C07314=1196.979,384.407,-79.887,-175.944,8.413,148.484
C07315=1196.984,384.160,-79.852,-175.945,8.410,148.484
C07316=1196.988,383.912,-79.818,-175.946,8.406,148.483
C07317=1196.992,383.664,-79.783,-175.947,8.404,148.483
C07318=1196.995,383.417,-79.748,-175.948,8.401,148.482
C07319=1197.000,383.170,-79.714,-175.948,8.397,148.481
C07320=1197.004,382.921,-79.679,-175.949,8.394,148.481
C07321=1197.007,382.674,-79.645,-175.950,8.392,148.480
C07322=1197.011,382.426,-79.610,-175.951,8.388,148.480
C07323=1197.016,382.179,-79.576,-175.952,8.385,148.479
C07324=1197.019,381.931,-79.541,-175.953,8.383,148.479
C07325=1197.024,381.684,-79.507,-175.954,8.379,148.478
C07326=1197.027,381.436,-79.471,-175.955,8.377,148.478
C07327=1197.031,381.189,-79.438,-175.956,8.374,148.477
C07328=1197.036,380.942,-79.403,-175.957,8.370,148.477
C07329=1197.040,380.693,-79.368,-175.958,8.368,148.476
C07330=1197.044,380.446,-79.334,-175.959,8.365,148.476
C07331=1197.048,380.198,-79.300,-175.960,8.362,148.475
C07332=1197.052,379.951,-79.265,-175.961,8.359,148.475
C07333=1197.055,379.703,-79.231,-175.962,8.356,148.474
C07334=1197.060,379.456,-79.196,-175.963,8.353,148.474
C07335=1197.065,379.208,-79.162,-175.965,8.349,148.473
C07336=1197.068,378.960,-79.128,-175.965,8.346,148.473
C07337=1197.072,378.713,-79.093,-175.967,8.343,148.472
C07338=1197.076,378.465,-79.058,-175.967,8.340,148.472
C07339=1197.080,378.218,-79.025,-175.969,8.337,148.471
C07340=1197.084,377.970,-78.990,-175.969,8.334,148.471
C07341=1197.088,377.722,-78.956,-175.971,8.331,148.470
C07342=1197.092,377.475,-78.921,-175.972,8.327,148.470
C07343=1197.096,377.227,-78.887,-175.973,8.325,148.469
C07344=1197.100,376.980,-78.853,-175.974,8.322,148.469
C07345=1197.104,376.732,-78.818,-175.975,8.319,148.468
C07346=1197.108,376.485,-78.784,-175.976,8.316,148.468
C07347=1197.113,376.237,-78.749,-175.978,8.312,148.467
C07348=1197.116,375.989,-78.716,-175.979,8.309,148.467
C07349=1197.121,375.741,-78.681,-175.980,8.306,148.467
C07350=1197.125,375.494,-78.648,-175.981,8.303,148.466
C07351=1197.129,375.246,-78.613,-175.983,8.300,148.466
C07352=1197.132,374.999,-78.579,-175.984,8.297,148.465
C07353=1197.136,374.751,-78.544,-175.985,8.294,148.465
C07354=1197.140,374.504,-78.510,-175.986,8.291,148.464
C07355=1197.145,374.256,-78.476,-175.988,8.287,148.464
C07356=1197.149,374.008,-78.442,-175.989,8.285,148.463
C07357=1197.153,373.760,-78.408,-175.990,8.281,148.463
C07358=1197.157,373.513,-78.374,-175.992,8.278,148.462
C07359=1197.161,373.265,-78.339,-175.993,8.275,148.462
C07360=1197.165,373.018,-78.306,-175.994,8.272,148.462
C07361=1197.169,372.770,-78.271,-175.995,8.268,148.461
C07362=1197.173,372.522,-78.237,-175.997,8.265,148.461
C07363=1197.177,372.275,-78.203,-175.998,8.263,148.460
C07364=1197.181,372.027,-78.170,-176.000,8.259,148.460
C07365=1197.185,371.779,-78.135,-176.001,8.256,148.459
C07366=1197.189,371.532,-78.101,-176.003,8.253,148.459
C07367=1197.194,371.285,-78.066,-176.003,8.249,148.458
C07368=1197.197,371.036,-78.033,-176.005,8.247,148.458
C07369=1197.201,370.789,-77.999,-176.006,8.243,148.457
C07370=1197.206,370.542,-77.965,-176.008,8.240,148.457
C07371=1197.210,370.294,-77.931,-176.009,8.237,148.457
C07372=1197.214,370.046,-77.897,-176.011,8.234,148.456
C07373=1197.218,369.799,-77.863,-176.012,8.231,148.456
C07374=1197.222,369.551,-77.829,-176.014,8.227,148.455
C07375=1197.226,369.303,-77.795,-176.015,8.225,148.455
C07376=1197.230,369.056,-77.761,-176.017,8.221,148.455
C07377=1197.234,368.808,-77.727,-176.018,8.218,148.454
C07378=1197.238,368.560,-77.693,-176.020,8.214,148.454
C07379=1197.242,368.312,-77.660,-176.021,8.212,148.453
C07380=1197.246,368.065,-77.625,-176.023,8.208,148.453
C07381=1197.250,367.818,-77.591,-176.024,8.205,148.453
C07382=1197.254,367.570,-77.558,-176.026,8.202,148.452
C07383=1197.258,367.322,-77.523,-176.027,8.199,148.452
C07384=1197.262,367.074,-77.490,-176.029,8.195,148.451
C07385=1197.267,366.793,-77.452,-176.030,8.192,148.451
C07386=1197.272,366.513,-77.413,-176.032,8.188,148.450
C07387=1197.277,366.232,-77.375,-176.034,8.184,148.450
C07388=1197.280,365.950,-77.337,-176.036,8.181,148.450
C07389=1197.285,365.703,-77.303,-176.037,8.178,148.449
C07390=1197.289,365.455,-77.270,-176.039,8.174,148.449
C07391=1197.293,365.208,-77.236,-176.040,8.172,148.449
C07392=1197.297,364.959,-77.202,-176.042,8.168,148.448
C07393=1197.301,364.712,-77.168,-176.044,8.164,148.448
C07394=1197.305,364.465,-77.135,-176.046,8.162,148.447
C07395=1197.309,364.217,-77.101,-176.048,8.158,148.447
C07396=1197.314,363.969,-77.067,-176.049,8.155,148.447
C07397=1197.317,363.721,-77.033,-176.051,8.152,148.446
C07398=1197.321,363.474,-77.000,-176.053,8.148,148.446
C07399=1197.325,363.226,-76.966,-176.054,8.146,148.446
C07400=1197.329,362.978,-76.933,-176.056,8.142,148.445
C07401=1197.334,362.731,-76.899,-176.057,8.140,148.445
C07402=1197.338,362.483,-76.866,-176.059,8.136,148.445
C07403=1197.342,362.235,-76.832,-176.061,8.132,148.444
C07404=1197.346,361.988,-76.798,-176.063,8.130,148.444
C07405=1197.350,361.740,-76.765,-176.064,8.126,148.443
C07406=1197.354,361.492,-76.732,-176.066,8.122,148.443
C07407=1197.358,361.245,-76.697,-176.068,8.120,148.443
C07408=1197.363,360.997,-76.664,-176.070,8.116,148.442
C07409=1197.366,360.749,-76.631,-176.071,8.113,148.442
C07410=1197.370,360.501,-76.598,-176.073,8.110,148.442
C07411=1197.374,360.254,-76.564,-176.075,8.107,148.441
C07412=1197.378,360.006,-76.531,-176.077,8.103,148.441
C07413=1197.382,359.758,-76.497,-176.078,8.100,148.441
C07414=1197.387,359.510,-76.464,-176.081,8.097,148.441
C07415=1197.391,359.263,-76.430,-176.082,8.093,148.440
C07416=1197.395,359.015,-76.396,-176.084,8.091,148.440
C07417=1197.399,358.767,-76.363,-176.086,8.087,148.439
C07418=1197.403,358.519,-76.330,-176.088,8.084,148.439
C07419=1197.407,358.272,-76.297,-176.089,8.081,148.439
C07420=1197.411,358.024,-76.264,-176.091,8.078,148.439
C07421=1197.415,357.776,-76.230,-176.093,8.074,148.438
C07422=1197.419,357.529,-76.197,-176.096,8.071,148.438
C07423=1197.424,357.281,-76.164,-176.097,8.068,148.438
C07424=1197.427,357.034,-76.130,-176.099,8.065,148.437
C07425=1197.431,356.786,-76.097,-176.101,8.061,148.437
C07426=1197.436,356.538,-76.064,-176.102,8.059,148.437
C07427=1197.440,356.291,-76.031,-176.105,8.055,148.437
C07428=1197.443,356.042,-75.997,-176.107,8.052,148.436
C07429=1197.447,355.794,-75.964,-176.109,8.048,148.436
C07430=1197.452,355.547,-75.931,-176.110,8.046,148.436
C07431=1197.456,355.299,-75.898,-176.113,8.042,148.435
C07432=1197.460,355.051,-75.865,-176.114,8.039,148.435
C07433=1197.464,354.803,-75.832,-176.116,8.036,148.435
C07434=1197.468,354.556,-75.798,-176.118,8.033,148.435
C07435=1197.472,354.308,-75.765,-176.120,8.029,148.434
C07436=1197.476,354.060,-75.732,-176.122,8.026,148.434
C07437=1197.481,353.813,-75.699,-176.124,8.024,148.434
C07438=1197.485,353.564,-75.666,-176.126,8.020,148.433
C07439=1197.489,353.316,-75.633,-176.128,8.017,148.433
C07440=1197.493,353.069,-75.600,-176.130,8.013,148.433
C07441=1197.497,352.821,-75.567,-176.132,8.011,148.433
C07442=1197.502,352.573,-75.534,-176.134,8.007,148.432
C07443=1197.506,352.326,-75.501,-176.136,8.004,148.432
C07444=1197.509,352.078,-75.468,-176.138,8.001,148.432
C07445=1197.513,351.830,-75.435,-176.140,7.998,148.432
C07446=1197.518,351.582,-75.403,-176.142,7.995,148.431
C07447=1197.522,351.334,-75.369,-176.144,7.991,148.431
C07448=1197.526,351.087,-75.336,-176.145,7.988,148.431
C07449=1197.530,350.839,-75.303,-176.148,7.985,148.431
C07450=1197.534,350.591,-75.270,-176.150,7.982,148.430
C07451=1197.539,350.343,-75.237,-176.152,7.978,148.430
C07452=1197.542,350.095,-75.205,-176.154,7.976,148.430
C07453=1197.546,349.848,-75.172,-176.156,7.972,148.430
C07454=1197.550,349.600,-75.139,-176.158,7.969,148.429
C07455=1197.555,349.352,-75.107,-176.160,7.966,148.429
C07456=1197.560,349.104,-75.073,-176.162,7.963,148.429
C07457=1197.563,348.857,-75.041,-176.164,7.960,148.429
C07458=1197.567,348.609,-75.008,-176.166,7.956,148.428
C07459=1197.571,348.361,-74.975,-176.168,7.954,148.428
C07460=1197.576,348.113,-74.942,-176.170,7.951,148.428
C07461=1197.580,347.865,-74.910,-176.172,7.947,148.428
C07462=1197.583,347.617,-74.877,-176.175,7.944,148.428
C07463=1197.588,347.370,-74.844,-176.176,7.941,148.427
C07464=1197.592,347.121,-74.811,-176.178,7.938,148.427
C07465=1197.596,346.874,-74.778,-176.180,7.934,148.427
C07466=1197.601,346.626,-74.747,-176.182,7.931,148.427
C07467=1197.605,346.379,-74.714,-176.184,7.929,148.426
C07468=1197.609,346.130,-74.681,-176.186,7.925,148.426
C07469=1197.612,345.883,-74.649,-176.189,7.922,148.426
C07470=1197.617,345.635,-74.615,-176.191,7.919,148.426
C07471=1197.621,345.387,-74.583,-176.192,7.916,148.426
C07472=1197.625,345.139,-74.550,-176.195,7.913,148.425
C07473=1197.630,344.892,-74.518,-176.197,7.909,148.425
C07474=1197.634,344.644,-74.485,-176.199,7.906,148.425
C07475=1197.638,344.396,-74.453,-176.201,7.904,148.425
C07476=1197.642,344.148,-74.421,-176.203,7.900,148.424
C07477=1197.646,343.900,-74.388,-176.206,7.897,148.424
C07478=1197.650,343.651,-74.355,-176.208,7.894,148.424
C07479=1197.654,343.405,-74.323,-176.210,7.891,148.424
C07480=1197.659,343.156,-74.291,-176.212,7.888,148.424
C07481=1197.662,342.909,-74.258,-176.214,7.885,148.424
C07482=1197.667,342.661,-74.226,-176.216,7.881,148.423
C07483=1197.671,342.412,-74.193,-176.218,7.879,148.423
C07484=1197.675,342.165,-74.161,-176.220,7.876,148.423
C07485=1197.680,341.917,-74.129,-176.222,7.872,148.423
C07486=1197.683,341.669,-74.097,-176.225,7.869,148.423
C07487=1197.687,341.421,-74.064,-176.227,7.867,148.423
C07488=1197.692,341.173,-74.031,-176.229,7.863,148.422
C07489=1197.697,340.895,-73.995,-176.231,7.860,148.422
C07490=1197.701,340.617,-73.958,-176.234,7.857,148.422
C07491=1197.706,340.338,-73.923,-176.236,7.853,148.422
C07492=1197.710,340.060,-73.887,-176.239,7.849,148.421
C07493=1197.715,339.812,-73.855,-176.241,7.846,148.421
C07494=1197.718,339.564,-73.822,-176.243,7.844,148.421
C07495=1197.723,339.316,-73.790,-176.245,7.840,148.421
C07496=1197.726,339.068,-73.758,-176.247,7.837,148.421
C07497=1197.731,338.820,-73.726,-176.250,7.834,148.421
C07498=1197.735,338.572,-73.694,-176.252,7.832,148.421
C07499=1197.739,338.324,-73.661,-176.254,7.828,148.420
C07500=1197.744,338.077,-73.629,-176.256,7.825,148.420
C07501=1197.748,337.829,-73.597,-176.258,7.822,148.420
C07502=1197.752,337.581,-73.565,-176.260,7.819,148.420
C07503=1197.756,337.332,-73.532,-176.263,7.816,148.420
C07504=1197.761,337.085,-73.501,-176.265,7.813,148.420
C07505=1197.765,336.837,-73.469,-176.267,7.809,148.419
C07506=1197.768,336.589,-73.436,-176.269,7.807,148.419
C07507=1197.772,336.341,-73.404,-176.272,7.804,148.419
C07508=1197.777,336.094,-73.372,-176.274,7.800,148.419
C07509=1197.781,335.846,-73.340,-176.276,7.797,148.419
C07510=1197.785,335.597,-73.308,-176.278,7.795,148.419
C07511=1197.790,335.350,-73.276,-176.280,7.792,148.419
C07512=1197.793,335.102,-73.244,-176.283,7.788,148.418
C07513=1197.798,334.853,-73.212,-176.285,7.785,148.418
C07514=1197.802,334.606,-73.181,-176.287,7.783,148.418
C07515=1197.806,334.358,-73.149,-176.289,7.779,148.418
C07516=1197.810,334.110,-73.116,-176.291,7.776,148.418
C07517=1197.815,333.862,-73.085,-176.294,7.773,148.418
C07518=1197.818,333.614,-73.053,-176.296,7.771,148.418
C07519=1197.823,333.366,-73.020,-176.298,7.768,148.418
C07520=1197.827,333.119,-72.989,-176.301,7.764,148.417
C07521=1197.831,332.870,-72.958,-176.303,7.761,148.417
C07522=1197.836,332.622,-72.926,-176.305,7.759,148.417
C07523=1197.840,332.374,-72.894,-176.307,7.755,148.417
C07524=1197.843,332.126,-72.862,-176.310,7.752,148.417
C07525=1197.848,331.879,-72.831,-176.312,7.749,148.417
C07526=1197.852,331.631,-72.798,-176.314,7.746,148.417
C07527=1197.856,331.383,-72.766,-176.317,7.743,148.417
C07528=1197.861,331.135,-72.736,-176.319,7.740,148.416
C07529=1197.864,330.887,-72.704,-176.321,7.737,148.416
C07530=1197.869,330.639,-72.672,-176.323,7.735,148.416
C07531=1197.873,330.391,-72.640,-176.325,7.731,148.416
C07532=1197.877,330.144,-72.608,-176.328,7.728,148.416
C07533=1197.881,329.895,-72.577,-176.330,7.725,148.416
C07534=1197.885,329.647,-72.545,-176.332,7.722,148.416
C07535=1197.890,329.399,-72.513,-176.335,7.719,148.416
C07536=1197.894,329.151,-72.481,-176.337,7.716,148.415
C07537=1197.898,328.903,-72.451,-176.340,7.713,148.415
C07538=1197.902,328.655,-72.419,-176.341,7.711,148.415
C07539=1197.906,328.408,-72.387,-176.344,7.708,148.415
C07540=1197.910,328.159,-72.356,-176.346,7.704,148.415
C07541=1197.915,327.912,-72.324,-176.349,7.701,148.415
C07542=1197.919,327.663,-72.292,-176.351,7.699,148.415
C07543=1197.923,327.415,-72.261,-176.353,7.696,148.415
C07544=1197.927,327.167,-72.230,-176.355,7.692,148.415
C07545=1197.931,326.919,-72.199,-176.358,7.690,148.415
C07546=1197.936,326.671,-72.167,-176.360,7.687,148.414
C07547=1197.939,326.423,-72.135,-176.363,7.684,148.414
C07548=1197.944,326.175,-72.104,-176.365,7.680,148.414
C07549=1197.948,325.927,-72.073,-176.367,7.678,148.414
C07550=1197.952,325.679,-72.042,-176.369,7.675,148.414
C07551=1197.957,325.431,-72.009,-176.372,7.672,148.414
C07552=1197.961,325.183,-71.979,-176.374,7.669,148.414
C07553=1197.965,324.935,-71.947,-176.376,7.666,148.414
C07554=1197.970,324.687,-71.916,-176.378,7.663,148.414
C07555=1197.974,324.439,-71.884,-176.381,7.660,148.414
C07556=1197.978,324.191,-71.853,-176.384,7.657,148.414
C07557=1197.982,323.943,-71.822,-176.385,7.654,148.414
C07558=1197.986,323.695,-71.791,-176.388,7.651,148.414
C07559=1197.991,323.448,-71.759,-176.390,7.648,148.413
C07560=1197.995,323.199,-71.728,-176.393,7.645,148.413
C07561=1197.999,322.952,-71.697,-176.395,7.643,148.413
C07562=1198.003,322.703,-71.666,-176.397,7.640,148.413
C07563=1198.008,322.455,-71.635,-176.400,7.637,148.413
C07564=1198.011,322.208,-71.604,-176.402,7.633,148.413
C07565=1198.015,321.960,-71.573,-176.404,7.631,148.413
C07566=1198.019,321.711,-71.542,-176.407,7.628,148.413
C07567=1198.024,321.464,-71.510,-176.409,7.625,148.413
C07568=1198.028,321.216,-71.479,-176.412,7.622,148.413
C07569=1198.032,320.967,-71.448,-176.414,7.619,148.413
C07570=1198.037,320.720,-71.417,-176.416,7.616,148.413
C07571=1198.041,320.471,-71.386,-176.419,7.613,148.413
C07572=1198.045,320.223,-71.355,-176.421,7.611,148.413
C07573=1198.050,319.975,-71.324,-176.424,7.608,148.413
C07574=1198.053,319.727,-71.292,-176.426,7.604,148.412
C07575=1198.057,319.479,-71.262,-176.428,7.601,148.412
C07576=1198.061,319.231,-71.231,-176.431,7.599,148.412
C07577=1198.066,318.983,-71.200,-176.433,7.596,148.412
C07578=1198.070,318.735,-71.169,-176.436,7.593,148.412
C07579=1198.074,318.487,-71.138,-176.438,7.590,148.412
C07580=1198.079,318.239,-71.107,-176.440,7.587,148.412
C07581=1198.083,317.991,-71.077,-176.443,7.584,148.412
C07582=1198.087,317.742,-71.046,-176.445,7.581,148.412
C07583=1198.091,317.494,-71.015,-176.447,7.579,148.412
C07584=1198.096,317.247,-70.983,-176.450,7.576,148.412
C07585=1198.100,316.998,-70.952,-176.452,7.573,148.412
C07586=1198.104,316.751,-70.922,-176.455,7.570,148.412
C07587=1198.108,316.503,-70.891,-176.457,7.567,148.412
C07588=1198.112,316.254,-70.860,-176.459,7.564,148.412
C07589=1198.117,316.006,-70.829,-176.462,7.561,148.412
C07590=1198.121,315.759,-70.799,-176.464,7.558,148.412
C07591=1198.125,315.510,-70.768,-176.466,7.555,148.412
C07592=1198.129,315.262,-70.737,-176.469,7.552,148.412
C07593=1198.134,314.986,-70.703,-176.472,7.549,148.412
C07594=1198.139,314.709,-70.669,-176.475,7.546,148.412
C07595=1198.143,314.433,-70.635,-176.477,7.543,148.411
C07596=1198.148,314.158,-70.601,-176.479,7.540,148.411
C07597=1198.152,313.909,-70.569,-176.482,7.537,148.411
C07598=1198.157,313.660,-70.539,-176.485,7.534,148.411
C07599=1198.161,313.413,-70.509,-176.487,7.531,148.411
C07600=1198.166,313.165,-70.478,-176.489,7.528,148.411
C07601=1198.170,312.916,-70.447,-176.492,7.525,148.411
C07602=1198.173,312.668,-70.417,-176.495,7.522,148.411
C07603=1198.178,312.420,-70.386,-176.497,7.520,148.411
C07604=1198.182,312.173,-70.356,-176.499,7.517,148.411
C07605=1198.186,311.924,-70.325,-176.502,7.514,148.411
C07606=1198.191,311.676,-70.294,-176.504,7.512,148.411
C07607=1198.195,311.428,-70.265,-176.506,7.509,148.411
C07608=1198.199,311.180,-70.234,-176.509,7.506,148.411
C07609=1198.203,310.931,-70.203,-176.511,7.502,148.411
C07610=1198.207,310.684,-70.173,-176.514,7.500,148.411
C07611=1198.212,310.436,-70.142,-176.516,7.497,148.411
C07612=1198.216,310.187,-70.113,-176.519,7.494,148.411
C07613=1198.221,309.939,-70.082,-176.521,7.492,148.411
C07614=1198.225,309.692,-70.052,-176.523,7.489,148.411
C07615=1198.229,309.443,-70.021,-176.526,7.486,148.411
C07616=1198.233,309.195,-69.991,-176.528,7.483,148.411
C07617=1198.237,308.947,-69.960,-176.531,7.480,148.411
C07618=1198.242,308.699,-69.930,-176.533,7.477,148.411
C07619=1198.246,308.451,-69.900,-176.536,7.474,148.411
C07620=1198.251,308.203,-69.869,-176.538,7.472,148.411
C07621=1198.254,307.954,-69.839,-176.541,7.469,148.411
C07622=1198.259,307.706,-69.809,-176.543,7.466,148.411
C07623=1198.263,307.458,-69.779,-176.545,7.464,148.411
C07624=1198.267,307.210,-69.748,-176.548,7.461,148.411
C07625=1198.272,306.962,-69.718,-176.551,7.458,148.411
C07626=1198.276,306.714,-69.688,-176.553,7.455,148.411
C07627=1198.280,306.466,-69.658,-176.555,7.452,148.411
C07628=1198.284,306.217,-69.628,-176.558,7.449,148.411
C07629=1198.289,305.969,-69.598,-176.560,7.447,148.411
C07630=1198.292,305.721,-69.567,-176.563,7.444,148.411
C07631=1198.297,305.473,-69.537,-176.565,7.441,148.411
C07632=1198.301,305.225,-69.507,-176.568,7.439,148.411
C07633=1198.306,304.976,-69.477,-176.570,7.436,148.411
C07634=1198.310,304.729,-69.447,-176.573,7.433,148.411
C07635=1198.314,304.480,-69.418,-176.576,7.430,148.411
C07636=1198.319,304.232,-69.387,-176.577,7.427,148.411
C07637=1198.323,303.984,-69.357,-176.580,7.424,148.411
C07638=1198.327,303.737,-69.327,-176.583,7.421,148.411
C07639=1198.332,303.488,-69.297,-176.585,7.419,148.411
C07640=1198.335,303.240,-69.267,-176.587,7.416,148.411
C07641=1198.340,302.991,-69.236,-176.590,7.413,148.411
C07642=1198.344,302.743,-69.207,-176.592,7.411,148.411
C07643=1198.348,302.495,-69.177,-176.595,7.408,148.411
C07644=1198.353,302.247,-69.147,-176.598,7.405,148.411
C07645=1198.357,301.998,-69.117,-176.600,7.402,148.411
C07646=1198.361,301.751,-69.087,-176.603,7.399,148.411
C07647=1198.365,301.502,-69.058,-176.605,7.396,148.411
C07648=1198.370,301.254,-69.028,-176.607,7.394,148.411
C07649=1198.374,301.006,-68.998,-176.610,7.391,148.411
C07650=1198.378,300.758,-68.968,-176.612,7.388,148.411
C07651=1198.382,300.510,-68.939,-176.614,7.386,148.411
C07652=1198.387,300.262,-68.908,-176.617,7.383,148.411
C07653=1198.391,300.013,-68.878,-176.620,7.380,148.411
C07654=1198.395,299.765,-68.849,-176.622,7.377,148.411
C07655=1198.400,299.517,-68.819,-176.625,7.374,148.411
C07656=1198.404,299.269,-68.789,-176.627,7.372,148.411
C07657=1198.408,299.021,-68.759,-176.630,7.369,148.411
C07658=1198.413,298.772,-68.730,-176.632,7.366,148.411
C07659=1198.417,298.524,-68.700,-176.634,7.364,148.411
C07660=1198.421,298.276,-68.671,-176.637,7.361,148.411
C07661=1198.426,298.027,-68.641,-176.640,7.358,148.411
C07662=1198.430,297.780,-68.611,-176.642,7.356,148.412
C07663=1198.434,297.531,-68.581,-176.645,7.353,148.412
C07664=1198.438,297.283,-68.552,-176.647,7.350,148.412
C07665=1198.443,297.035,-68.523,-176.649,7.348,148.412
C07666=1198.447,296.787,-68.493,-176.652,7.345,148.412
C07667=1198.451,296.539,-68.464,-176.655,7.342,148.412
C07668=1198.456,296.290,-68.434,-176.657,7.339,148.412
C07669=1198.460,296.042,-68.404,-176.660,7.336,148.412
C07670=1198.465,295.794,-68.375,-176.662,7.334,148.412
C07671=1198.469,295.546,-68.345,-176.665,7.331,148.412
C07672=1198.473,295.297,-68.316,-176.667,7.328,148.412
C07673=1198.477,295.049,-68.286,-176.669,7.326,148.412
C07674=1198.481,294.801,-68.257,-176.672,7.323,148.412
C07675=1198.485,294.552,-68.228,-176.675,7.320,148.412
C07676=1198.490,294.304,-68.198,-176.677,7.318,148.412
C07677=1198.494,294.057,-68.169,-176.680,7.315,148.412
C07678=1198.499,293.808,-68.140,-176.683,7.312,148.412
C07679=1198.503,293.560,-68.110,-176.685,7.310,148.412
C07680=1198.507,293.312,-68.081,-176.688,7.307,148.412
C07681=1198.511,293.064,-68.051,-176.690,7.305,148.412
C07682=1198.515,292.815,-68.022,-176.692,7.302,148.413
C07683=1198.519,292.567,-67.992,-176.695,7.299,148.413
C07684=1198.524,292.319,-67.963,-176.697,7.296,148.413
C07685=1198.529,292.071,-67.934,-176.700,7.293,148.413
C07686=1198.533,291.822,-67.905,-176.702,7.291,148.413
C07687=1198.537,291.574,-67.876,-176.705,7.288,148.413
C07688=1198.541,291.326,-67.846,-176.708,7.285,148.413
C07689=1198.545,291.078,-67.817,-176.710,7.283,148.413
C07690=1198.550,290.829,-67.788,-176.712,7.280,148.413
C07691=1198.555,290.581,-67.759,-176.715,7.277,148.413
C07692=1198.559,290.333,-67.729,-176.717,7.275,148.413
C07693=1198.563,290.085,-67.700,-176.720,7.272,148.413
C07694=1198.567,289.836,-67.670,-176.723,7.270,148.413
C07695=1198.572,289.587,-67.642,-176.725,7.267,148.413
C07696=1198.577,289.340,-67.613,-176.728,7.264,148.413
C07697=1198.581,289.065,-67.581,-176.731,7.261,148.413
C07698=1198.585,288.791,-67.548,-176.733,7.258,148.413
C07699=1198.590,288.517,-67.517,-176.736,7.256,148.414
C07700=1198.596,288.242,-67.484,-176.739,7.253,148.414
C07701=1198.600,287.994,-67.455,-176.741,7.250,148.414
C07702=1198.603,287.746,-67.426,-176.744,7.247,148.414
C07703=1198.608,287.497,-67.397,-176.746,7.245,148.414
C07704=1198.612,287.249,-67.368,-176.749,7.242,148.414
C07705=1198.617,287.000,-67.340,-176.751,7.240,148.414
C07706=1198.621,286.752,-67.310,-176.754,7.237,148.414
C07707=1198.625,286.505,-67.282,-176.757,7.234,148.414
C07708=1198.630,286.256,-67.253,-176.759,7.232,148.414
C07709=1198.634,286.008,-67.223,-176.762,7.229,148.414
C07710=1198.638,285.759,-67.195,-176.764,7.227,148.414
C07711=1198.643,285.511,-67.166,-176.767,7.224,148.414
C07712=1198.647,285.263,-67.137,-176.769,7.221,148.414
C07713=1198.651,285.014,-67.108,-176.771,7.218,148.414
C07714=1198.656,284.766,-67.080,-176.775,7.216,148.415
C07715=1198.660,284.518,-67.050,-176.777,7.213,148.415
C07716=1198.664,284.269,-67.022,-176.779,7.210,148.415
C07717=1198.668,284.021,-66.993,-176.782,7.208,148.415
C07718=1198.673,283.773,-66.964,-176.784,7.205,148.415
C07719=1198.678,283.525,-66.935,-176.786,7.203,148.415
C07720=1198.681,283.276,-66.907,-176.790,7.200,148.415
C07721=1198.686,283.028,-66.878,-176.792,7.197,148.415
C07722=1198.691,282.780,-66.849,-176.794,7.195,148.415
C07723=1198.694,282.531,-66.821,-176.797,7.192,148.415
C07724=1198.699,282.283,-66.792,-176.799,7.190,148.415
C07725=1198.704,282.035,-66.763,-176.802,7.187,148.415
C07726=1198.708,281.787,-66.735,-176.805,7.185,148.416
C07727=1198.712,281.538,-66.706,-176.807,7.182,148.416
C07728=1198.717,281.290,-66.677,-176.810,7.179,148.416
C07729=1198.721,281.042,-66.649,-176.812,7.177,148.416
C07730=1198.725,280.793,-66.620,-176.815,7.174,148.416
C07731=1198.729,280.545,-66.591,-176.817,7.172,148.416
C07732=1198.734,280.297,-66.563,-176.820,7.169,148.416
C07733=1198.738,280.048,-66.534,-176.822,7.167,148.416
C07734=1198.743,279.800,-66.507,-176.825,7.164,148.416
C07735=1198.747,279.552,-66.477,-176.827,7.162,148.416
C07736=1198.751,279.303,-66.449,-176.830,7.159,148.417
C07737=1198.756,279.055,-66.421,-176.832,7.157,148.417
C07738=1198.760,278.806,-66.392,-176.835,7.154,148.417
C07739=1198.765,278.558,-66.364,-176.837,7.152,148.417
C07740=1198.769,278.310,-66.335,-176.840,7.149,148.417
C07741=1198.773,278.061,-66.307,-176.843,7.146,148.417
C07742=1198.778,277.813,-66.278,-176.845,7.144,148.417
C07743=1198.781,277.565,-66.250,-176.848,7.141,148.417
C07744=1198.787,277.316,-66.222,-176.850,7.139,148.417
C07745=1198.790,277.068,-66.193,-176.853,7.136,148.418
C07746=1198.795,276.820,-66.165,-176.856,7.134,148.418
C07747=1198.799,276.571,-66.137,-176.858,7.131,148.418
C07748=1198.804,276.323,-66.108,-176.860,7.128,148.418
C07749=1198.808,276.075,-66.080,-176.864,7.126,148.418
C07750=1198.811,275.826,-66.052,-176.866,7.124,148.418
C07751=1198.816,275.578,-66.023,-176.868,7.121,148.418
C07752=1198.820,275.330,-65.995,-176.871,7.118,148.418
C07753=1198.825,275.081,-65.967,-176.874,7.116,148.418
C07754=1198.829,274.833,-65.939,-176.876,7.114,148.419
C07755=1198.834,274.585,-65.910,-176.879,7.111,148.419
C07756=1198.838,274.336,-65.882,-176.881,7.108,148.419
C07757=1198.842,274.088,-65.854,-176.884,7.106,148.419
C07758=1198.847,273.839,-65.826,-176.886,7.104,148.419
C07759=1198.851,273.591,-65.798,-176.889,7.100,148.419
C07760=1198.856,273.342,-65.770,-176.891,7.098,148.419
C07761=1198.860,273.094,-65.742,-176.894,7.096,148.419
C07762=1198.864,272.845,-65.714,-176.896,7.093,148.419
C07763=1198.869,272.597,-65.685,-176.899,7.090,148.419
C07764=1198.873,272.349,-65.658,-176.901,7.088,148.420
C07765=1198.877,272.101,-65.630,-176.904,7.086,148.420
C07766=1198.882,271.853,-65.601,-176.906,7.083,148.420
C07767=1198.886,271.604,-65.573,-176.909,7.080,148.420
C07768=1198.891,271.355,-65.546,-176.912,7.079,148.420
C07769=1198.895,271.107,-65.517,-176.914,7.076,148.420
C07770=1198.900,270.859,-65.489,-176.917,7.073,148.420
C07771=1198.903,270.610,-65.461,-176.920,7.071,148.421
C07772=1198.908,270.362,-65.433,-176.922,7.068,148.421
C07773=1198.913,270.113,-65.406,-176.925,7.065,148.421
C07774=1198.917,269.865,-65.378,-176.927,7.063,148.421
C07775=1198.921,269.617,-65.350,-176.930,7.061,148.421
C07776=1198.926,269.368,-65.321,-176.932,7.058,148.421
C07777=1198.930,269.120,-65.294,-176.935,7.055,148.421
C07778=1198.935,268.872,-65.266,-176.937,7.054,148.421
C07779=1198.938,268.623,-65.238,-176.940,7.051,148.422
C07780=1198.944,268.374,-65.211,-176.942,7.048,148.422
C07781=1198.948,268.127,-65.183,-176.945,7.047,148.422
C07782=1198.952,267.878,-65.155,-176.948,7.044,148.422
C07783=1198.957,267.629,-65.128,-176.950,7.041,148.422
C07784=1198.960,267.381,-65.099,-176.953,7.039,148.422
C07785=1198.965,267.133,-65.071,-176.955,7.037,148.422
C07786=1198.970,266.884,-65.044,-176.958,7.034,148.422
C07787=1198.974,266.636,-65.016,-176.960,7.032,148.423
C07788=1198.978,266.387,-64.989,-176.963,7.029,148.423
C07789=1198.983,266.139,-64.961,-176.965,7.026,148.423
C07790=1198.987,265.891,-64.933,-176.968,7.024,148.423
C07791=1198.991,265.642,-64.906,-176.971,7.022,148.423
C07792=1198.996,265.394,-64.877,-176.973,7.019,148.423
C07793=1199.000,265.145,-64.850,-176.976,7.017,148.424
C07794=1199.005,264.897,-64.822,-176.978,7.015,148.424
C07795=1199.009,264.648,-64.795,-176.981,7.012,148.424
C07796=1199.014,264.401,-64.767,-176.983,7.010,148.424
C07797=1199.018,264.151,-64.740,-176.986,7.007,148.424
C07798=1199.022,263.903,-64.712,-176.988,7.005,148.424
C07799=1199.027,263.655,-64.685,-176.991,7.002,148.424
C07800=1199.031,263.406,-64.658,-176.994,7.000,148.424
C07801=1199.036,263.133,-64.627,-176.997,6.997,148.425
C07802=1199.041,262.861,-64.597,-176.999,6.995,148.425
C07803=1199.045,262.587,-64.567,-177.002,6.992,148.425
C07804=1199.051,262.315,-64.537,-177.005,6.989,148.425
C07805=1199.055,262.067,-64.509,-177.007,6.987,148.425
C07806=1199.059,261.818,-64.481,-177.010,6.984,148.425
C07807=1199.064,261.569,-64.454,-177.012,6.982,148.426
C07808=1199.068,261.321,-64.427,-177.015,6.979,148.426
C07809=1199.073,261.073,-64.400,-177.018,6.977,148.426
C07810=1199.077,260.824,-64.372,-177.020,6.974,148.426
C07811=1199.081,260.576,-64.344,-177.023,6.972,148.426
C07812=1199.086,260.327,-64.317,-177.025,6.970,148.426
C07813=1199.090,260.079,-64.290,-177.028,6.968,148.427
C07814=1199.095,259.830,-64.263,-177.030,6.965,148.427
C07815=1199.099,259.582,-64.235,-177.033,6.962,148.427
C07816=1199.103,259.333,-64.208,-177.036,6.961,148.427
C07817=1199.108,259.085,-64.181,-177.038,6.958,148.427
C07818=1199.113,258.836,-64.154,-177.041,6.956,148.427
C07819=1199.117,258.588,-64.127,-177.043,6.953,148.427
C07820=1199.120,258.340,-64.099,-177.046,6.951,148.428
C07821=1199.125,258.091,-64.072,-177.049,6.949,148.428
C07822=1199.130,257.843,-64.045,-177.051,6.946,148.428
C07823=1199.134,257.594,-64.018,-177.054,6.944,148.428
C07824=1199.139,257.346,-63.991,-177.056,6.942,148.428
C07825=1199.144,257.097,-63.964,-177.059,6.939,148.429
C07826=1199.147,256.848,-63.936,-177.061,6.937,148.429
C07827=1199.151,256.600,-63.909,-177.064,6.935,148.429
C07828=1199.156,256.352,-63.882,-177.067,6.932,148.429
C07829=1199.161,256.103,-63.855,-177.069,6.930,148.429
C07830=1199.165,255.855,-63.828,-177.072,6.928,148.429
C07831=1199.170,255.606,-63.801,-177.074,6.925,148.429
C07832=1199.175,255.358,-63.774,-177.077,6.923,148.430
C07833=1199.178,255.109,-63.747,-177.080,6.920,148.430
C07834=1199.183,254.860,-63.720,-177.082,6.918,148.430
C07835=1199.187,254.612,-63.693,-177.084,6.916,148.430
C07836=1199.192,254.363,-63.666,-177.087,6.913,148.430
C07837=1199.196,254.115,-63.640,-177.090,6.911,148.431
C07838=1199.200,253.867,-63.612,-177.092,6.909,148.431
C07839=1199.205,253.618,-63.585,-177.095,6.906,148.431
C07840=1199.210,253.370,-63.558,-177.097,6.904,148.431
C07841=1199.214,253.122,-63.532,-177.100,6.902,148.431
C07842=1199.218,252.872,-63.504,-177.103,6.899,148.431
C07843=1199.222,252.624,-63.477,-177.105,6.897,148.432
C07844=1199.227,252.375,-63.450,-177.108,6.894,148.432
C07845=1199.231,252.127,-63.424,-177.111,6.893,148.432
C07846=1199.236,251.879,-63.397,-177.113,6.890,148.432
C07847=1199.241,251.630,-63.370,-177.116,6.888,148.432
C07848=1199.245,251.381,-63.344,-177.118,6.886,148.432
C07849=1199.249,251.133,-63.317,-177.121,6.884,148.433
C07850=1199.254,250.884,-63.290,-177.123,6.881,148.433
C07851=1199.258,250.636,-63.263,-177.126,6.879,148.433
C07852=1199.262,250.388,-63.236,-177.128,6.877,148.433
C07853=1199.267,250.139,-63.210,-177.131,6.874,148.433
C07854=1199.271,249.890,-63.184,-177.133,6.872,148.434
C07855=1199.276,249.642,-63.156,-177.136,6.870,148.434
C07856=1199.281,249.393,-63.129,-177.139,6.867,148.434
C07857=1199.285,249.145,-63.103,-177.141,6.865,148.434
C07858=1199.289,248.896,-63.077,-177.144,6.863,148.434
C07859=1199.293,248.648,-63.050,-177.146,6.860,148.434
C07860=1199.298,248.399,-63.023,-177.149,6.858,148.435
C07861=1199.303,248.150,-62.997,-177.151,6.856,148.435
C07862=1199.307,247.902,-62.970,-177.154,6.853,148.435
C07863=1199.312,247.654,-62.943,-177.156,6.851,148.435
C07864=1199.316,247.405,-62.917,-177.159,6.849,148.436
C07865=1199.320,247.156,-62.890,-177.162,6.846,148.436
C07866=1199.324,246.908,-62.864,-177.164,6.844,148.436
C07867=1199.329,246.659,-62.838,-177.167,6.843,148.436
C07868=1199.333,246.411,-62.811,-177.170,6.840,148.436
C07869=1199.338,246.162,-62.784,-177.172,6.838,148.437
C07870=1199.343,245.913,-62.758,-177.175,6.836,148.437
C07871=1199.347,245.665,-62.731,-177.177,6.834,148.437
C07872=1199.352,245.416,-62.705,-177.180,6.831,148.437
C07873=1199.356,245.168,-62.678,-177.183,6.829,148.437
C07874=1199.360,244.920,-62.652,-177.185,6.827,148.437
C07875=1199.365,244.671,-62.626,-177.188,6.824,148.438
C07876=1199.368,244.422,-62.599,-177.190,6.822,148.438
C07877=1199.374,244.174,-62.573,-177.193,6.820,148.438
C07878=1199.378,243.926,-62.547,-177.195,6.817,148.438
C07879=1199.383,243.677,-62.520,-177.198,6.815,148.439
C07880=1199.387,243.428,-62.494,-177.201,6.813,148.439
C07881=1199.392,243.179,-62.468,-177.203,6.811,148.439
C07882=1199.396,242.931,-62.441,-177.206,6.809,148.439
C07883=1199.400,242.682,-62.415,-177.208,6.806,148.439
C07884=1199.405,242.433,-62.389,-177.211,6.805,148.440
C07885=1199.409,242.185,-62.363,-177.214,6.802,148.440
C07886=1199.414,241.936,-62.336,-177.216,6.800,148.440
C07887=1199.418,241.688,-62.310,-177.218,6.798,148.440
C07888=1199.423,241.440,-62.284,-177.221,6.796,148.440
C07889=1199.428,241.191,-62.258,-177.224,6.793,148.441
C07890=1199.431,240.942,-62.232,-177.226,6.791,148.441
C07891=1199.436,240.694,-62.206,-177.229,6.789,148.441
C07892=1199.440,240.445,-62.179,-177.232,6.786,148.441
C07893=1199.445,240.196,-62.153,-177.234,6.784,148.441
C07894=1199.449,239.948,-62.128,-177.236,6.782,148.442
C07895=1199.454,239.700,-62.101,-177.239,6.780,148.442
C07896=1199.458,239.451,-62.075,-177.242,6.778,148.442
C07897=1199.462,239.202,-62.049,-177.244,6.775,148.442
C07898=1199.467,238.953,-62.023,-177.247,6.774,148.443
C07899=1199.472,238.705,-61.997,-177.249,6.771,148.443
C07900=1199.476,238.457,-61.971,-177.252,6.769,148.443
C07901=1199.481,238.207,-61.944,-177.255,6.767,148.443
C07902=1199.485,237.959,-61.919,-177.257,6.765,148.443
C07903=1199.489,237.711,-61.892,-177.260,6.763,148.444
C07904=1199.494,237.462,-61.867,-177.263,6.760,148.444
C07905=1199.500,237.190,-61.838,-177.265,6.758,148.444
C07906=1199.504,236.919,-61.809,-177.268,6.755,148.444
C07907=1199.509,236.647,-61.781,-177.271,6.754,148.445
C07908=1199.514,236.376,-61.754,-177.274,6.751,148.445
C07909=1199.518,236.128,-61.727,-177.276,6.749,148.445
C07910=1199.522,235.879,-61.702,-177.279,6.747,148.445
C07911=1199.528,235.630,-61.676,-177.282,6.744,148.445
C07912=1199.532,235.382,-61.650,-177.284,6.742,148.446
C07913=1199.536,235.133,-61.624,-177.287,6.740,148.446
C07914=1199.540,234.884,-61.598,-177.289,6.738,148.446
C07915=1199.545,234.636,-61.573,-177.292,6.735,148.447
C07916=1199.549,234.387,-61.547,-177.295,6.733,148.447
C07917=1199.554,234.138,-61.521,-177.297,6.731,148.447
C07918=1199.559,233.889,-61.495,-177.300,6.730,148.447
C07919=1199.563,233.641,-61.470,-177.302,6.727,148.447
C07920=1199.568,233.392,-61.444,-177.305,6.725,148.448
C07921=1199.572,233.143,-61.418,-177.308,6.723,148.448
C07922=1199.577,232.895,-61.393,-177.310,6.721,148.448
C07923=1199.581,232.647,-61.367,-177.313,6.719,148.448
C07924=1199.585,232.398,-61.341,-177.316,6.716,148.449
C07925=1199.590,232.149,-61.315,-177.318,6.714,148.449
C07926=1199.595,231.901,-61.290,-177.321,6.712,148.449
C07927=1199.599,231.652,-61.264,-177.323,6.710,148.449
C07928=1199.603,231.403,-61.238,-177.325,6.708,148.450
C07929=1199.608,231.155,-61.213,-177.329,6.706,148.450
C07930=1199.612,230.906,-61.187,-177.331,6.703,148.450
C07931=1199.617,230.657,-61.161,-177.333,6.702,148.450
C07932=1199.621,230.409,-61.136,-177.336,6.700,148.451
C07933=1199.626,230.160,-61.111,-177.338,6.698,148.451
C07934=1199.630,229.911,-61.085,-177.341,6.695,148.451
C07935=1199.635,229.663,-61.060,-177.344,6.693,148.451
C07936=1199.639,229.414,-61.034,-177.347,6.691,148.452
C07937=1199.644,229.166,-61.008,-177.349,6.689,148.452
C07938=1199.648,228.917,-60.983,-177.351,6.687,148.452
C07939=1199.653,228.668,-60.958,-177.355,6.685,148.452
C07940=1199.658,228.420,-60.932,-177.357,6.682,148.452
C07941=1199.662,228.171,-60.907,-177.359,6.681,148.453
C07942=1199.666,227.922,-60.881,-177.362,6.679,148.453
C07943=1199.671,227.673,-60.856,-177.364,6.677,148.453
C07944=1199.675,227.424,-60.830,-177.367,6.674,148.453
C07945=1199.680,227.176,-60.805,-177.370,6.672,148.454
C07946=1199.684,226.927,-60.779,-177.372,6.670,148.454
C07947=1199.689,226.678,-60.754,-177.375,6.668,148.454
C07948=1199.693,226.430,-60.729,-177.378,6.666,148.455
C07949=1199.697,226.181,-60.704,-177.381,6.664,148.455
C07950=1199.702,225.933,-60.679,-177.383,6.661,148.455
C07951=1199.707,225.684,-60.653,-177.386,6.660,148.455
C07952=1199.712,225.436,-60.628,-177.388,6.658,148.456
C07953=1199.716,225.186,-60.603,-177.390,6.656,148.456
C07954=1199.721,224.938,-60.577,-177.393,6.654,148.456
C07955=1199.725,224.689,-60.552,-177.396,6.651,148.456
C07956=1199.729,224.440,-60.527,-177.399,6.649,148.457
C07957=1199.734,224.192,-60.502,-177.401,6.647,148.457
C07958=1199.738,223.943,-60.477,-177.404,6.645,148.457
C07959=1199.743,223.695,-60.451,-177.406,6.643,148.457
C07960=1199.748,223.445,-60.426,-177.409,6.640,148.458
C07961=1199.752,223.197,-60.401,-177.412,6.639,148.458
C07962=1199.756,222.949,-60.376,-177.414,6.637,148.458
C07963=1199.761,222.700,-60.351,-177.417,6.635,148.459
C07964=1199.765,222.451,-60.325,-177.419,6.633,148.459
C07965=1199.770,222.202,-60.301,-177.422,6.631,148.459
C07966=1199.775,221.954,-60.275,-177.425,6.628,148.459
C07967=1199.779,221.705,-60.251,-177.428,6.626,148.460
C07968=1199.784,221.456,-60.226,-177.430,6.624,148.460
C07969=1199.788,221.208,-60.201,-177.432,6.622,148.460
C07970=1199.793,220.958,-60.176,-177.435,6.621,148.460
C07971=1199.797,220.711,-60.151,-177.438,6.619,148.461
C07972=1199.802,220.461,-60.126,-177.440,6.617,148.461
C07973=1199.806,220.213,-60.100,-177.443,6.614,148.461
C07974=1199.810,219.964,-60.076,-177.446,6.612,148.461
C07975=1199.815,219.715,-60.051,-177.448,6.610,148.462
C07976=1199.820,219.467,-60.026,-177.450,6.608,148.462
C07977=1199.825,219.218,-60.001,-177.453,6.606,148.462
C07978=1199.829,218.970,-59.976,-177.456,6.605,148.463
C07979=1199.833,218.720,-59.951,-177.459,6.602,148.463
C07980=1199.838,218.472,-59.926,-177.462,6.600,148.463
C07981=1199.842,218.223,-59.902,-177.464,6.598,148.463
C07982=1199.847,217.974,-59.876,-177.466,6.596,148.464
C07983=1199.851,217.725,-59.852,-177.469,6.594,148.464
C07984=1199.856,217.477,-59.827,-177.472,6.592,148.464
C07985=1199.861,217.229,-59.802,-177.474,6.590,148.464
C07986=1199.865,216.979,-59.778,-177.477,6.588,148.465
C07987=1199.870,216.731,-59.753,-177.480,6.586,148.465
C07988=1199.874,216.481,-59.728,-177.482,6.584,148.465
C07989=1199.878,216.233,-59.703,-177.485,6.582,148.466
C07990=1199.883,215.985,-59.678,-177.487,6.580,148.466
C07991=1199.887,215.736,-59.654,-177.490,6.578,148.466
C07992=1199.892,215.487,-59.629,-177.492,6.576,148.466
C07993=1199.897,215.238,-59.605,-177.495,6.574,148.467
C07994=1199.901,214.990,-59.579,-177.498,6.572,148.467
C07995=1199.906,214.741,-59.555,-177.501,6.570,148.467
C07996=1199.910,214.492,-59.530,-177.503,6.568,148.468
C07997=1199.915,214.243,-59.506,-177.506,6.566,148.468
C07998=1199.919,213.995,-59.482,-177.508,6.564,148.468
C07999=1199.924,213.745,-59.457,-177.511,6.562,148.469
C08000=1199.928,213.497,-59.432,-177.513,6.560,148.469
C08001=1199.933,213.248,-59.408,-177.516,6.558,148.469
C08002=1199.937,212.999,-59.383,-177.519,6.556,148.469
C08003=1199.942,212.751,-59.358,-177.522,6.554,148.470
C08004=1199.946,212.503,-59.334,-177.524,6.552,148.470
C08005=1199.951,212.253,-59.309,-177.527,6.550,148.470
C08006=1199.955,212.005,-59.285,-177.529,6.548,148.470
C08007=1199.961,211.756,-59.260,-177.532,6.546,148.471
C08008=1199.965,211.508,-59.236,-177.535,6.544,148.471
C08009=1199.970,211.236,-59.210,-177.538,6.542,148.471
C08010=1199.975,210.966,-59.183,-177.540,6.540,148.472
C08011=1199.980,210.696,-59.156,-177.543,6.538,148.472
C08012=1199.985,210.426,-59.130,-177.546,6.535,148.472
C08013=1199.989,210.176,-59.105,-177.549,6.534,148.473
C08014=1199.993,209.928,-59.081,-177.552,6.532,148.473
C08015=1199.999,209.679,-59.056,-177.554,6.530,148.473
C08016=1200.003,209.431,-59.032,-177.556,6.528,148.474
C08017=1200.007,209.181,-59.009,-177.559,6.526,148.474
C08018=1200.012,208.932,-58.984,-177.562,6.524,148.474
C08019=1200.017,208.684,-58.960,-177.564,6.522,148.475
C08020=1200.022,208.435,-58.935,-177.567,6.521,148.475
C08021=1200.026,208.186,-58.911,-177.570,6.518,148.475
C08022=1200.030,207.938,-58.887,-177.573,6.516,148.476
C08023=1200.035,207.689,-58.862,-177.575,6.514,148.476
C08024=1200.040,207.440,-58.839,-177.578,6.512,148.476
C08025=1200.044,207.191,-58.814,-177.580,6.510,148.476
C08026=1200.049,206.942,-58.789,-177.583,6.508,148.477
C08027=1200.053,206.694,-58.765,-177.586,6.507,148.477
C08028=1200.057,206.445,-58.741,-177.588,6.505,148.477
C08029=1200.063,206.196,-58.717,-177.591,6.503,148.478
C08030=1200.067,205.947,-58.693,-177.593,6.501,148.478
C08031=1200.071,205.698,-58.669,-177.596,6.499,148.478
C08032=1200.075,205.450,-58.645,-177.598,6.497,148.478
C08033=1200.081,205.201,-58.621,-177.601,6.495,148.479
C08034=1200.085,204.952,-58.597,-177.604,6.494,148.479
C08035=1200.090,204.704,-58.573,-177.606,6.492,148.480
C08036=1200.094,204.454,-58.549,-177.610,6.489,148.480
C08037=1200.099,204.205,-58.524,-177.612,6.487,148.480
C08038=1200.103,203.957,-58.500,-177.614,6.485,148.480
C08039=1200.108,203.708,-58.477,-177.617,6.483,148.481
C08040=1200.112,203.460,-58.453,-177.620,6.482,148.481
C08041=1200.118,203.211,-58.428,-177.622,6.480,148.481
C08042=1200.122,202.961,-58.404,-177.625,6.478,148.482
C08043=1200.126,202.713,-58.380,-177.628,6.476,148.482
C08044=1200.130,202.464,-58.356,-177.630,6.474,148.482
C08045=1200.135,202.215,-58.333,-177.633,6.472,148.483
C08046=1200.140,201.967,-58.309,-177.636,6.471,148.483
C08047=1200.145,201.718,-58.285,-177.638,6.468,148.483
C08048=1200.149,201.469,-58.261,-177.640,6.467,148.483
C08049=1200.154,201.220,-58.237,-177.643,6.465,148.484
C08050=1200.158,200.971,-58.213,-177.646,6.463,148.484
C08051=1200.163,200.722,-58.190,-177.648,6.461,148.485
C08052=1200.167,200.474,-58.166,-177.651,6.459,148.485
C08053=1200.172,200.224,-58.142,-177.654,6.458,148.485
C08054=1200.176,199.976,-58.118,-177.656,6.456,148.486
C08055=1200.181,199.727,-58.094,-177.659,6.454,148.486
C08056=1200.186,199.478,-58.070,-177.662,6.452,148.486
C08057=1200.191,199.229,-58.047,-177.664,6.450,148.486
C08058=1200.195,198.981,-58.023,-177.666,6.448,148.487
C08059=1200.200,198.732,-57.999,-177.669,6.446,148.487
C08060=1200.204,198.483,-57.975,-177.672,6.444,148.487
C08061=1200.209,198.234,-57.952,-177.674,6.443,148.488
C08062=1200.213,197.985,-57.929,-177.677,6.441,148.488
C08063=1200.218,197.737,-57.904,-177.680,6.439,148.488
C08064=1200.222,197.487,-57.881,-177.682,6.437,148.489
C08065=1200.226,197.239,-57.857,-177.685,6.435,148.489
C08066=1200.231,196.990,-57.833,-177.688,6.434,148.489
C08067=1200.236,196.741,-57.810,-177.690,6.432,148.490
C08068=1200.240,196.492,-57.786,-177.693,6.430,148.490
C08069=1200.245,196.243,-57.762,-177.696,6.428,148.491
C08070=1200.250,195.994,-57.739,-177.698,6.426,148.491
C08071=1200.254,195.746,-57.715,-177.700,6.424,148.491
C08072=1200.259,195.497,-57.692,-177.703,6.422,148.491
C08073=1200.263,195.248,-57.668,-177.706,6.421,148.492
C08074=1200.268,194.999,-57.645,-177.708,6.419,148.492
C08075=1200.272,194.750,-57.621,-177.711,6.417,148.492
C08076=1200.277,194.501,-57.598,-177.714,6.415,148.493
C08077=1200.282,194.252,-57.574,-177.716,6.413,148.493
C08078=1200.287,194.003,-57.551,-177.719,6.411,148.493
C08079=1200.291,193.755,-57.527,-177.722,6.410,148.494
C08080=1200.296,193.506,-57.504,-177.724,6.408,148.494
C08081=1200.301,193.257,-57.480,-177.727,6.406,148.494
C08082=1200.306,193.008,-57.457,-177.730,6.404,148.495
C08083=1200.310,192.760,-57.434,-177.732,6.402,148.495
C08084=1200.314,192.511,-57.411,-177.735,6.401,148.495
C08085=1200.319,192.262,-57.387,-177.738,6.399,148.496
C08086=1200.323,192.013,-57.363,-177.740,6.397,148.496
C08087=1200.328,191.764,-57.340,-177.743,6.395,148.497
C08088=1200.333,191.515,-57.317,-177.746,6.393,148.497
C08089=1200.337,191.266,-57.293,-177.748,6.392,148.497
C08090=1200.341,191.017,-57.271,-177.751,6.390,148.498
C08091=1200.346,190.768,-57.247,-177.754,6.388,148.498
C08092=1200.351,190.519,-57.224,-177.756,6.386,148.498
C08093=1200.356,190.270,-57.201,-177.759,6.384,148.499
C08094=1200.361,190.022,-57.178,-177.761,6.382,148.499
C08095=1200.366,189.773,-57.154,-177.764,6.380,148.499
C08096=1200.370,189.524,-57.131,-177.766,6.379,148.499
C08097=1200.374,189.275,-57.108,-177.769,6.377,148.500
C08098=1200.379,189.026,-57.085,-177.772,6.375,148.500
C08099=1200.384,188.777,-57.061,-177.774,6.373,148.501
C08100=1200.388,188.528,-57.038,-177.777,6.371,148.501
C08101=1200.392,188.279,-57.015,-177.780,6.369,148.501
C08102=1200.398,188.031,-56.992,-177.782,6.368,148.502
C08103=1200.402,187.782,-56.969,-177.785,6.366,148.502
C08104=1200.407,187.533,-56.946,-177.787,6.365,148.502
C08105=1200.411,187.284,-56.923,-177.790,6.363,148.503
C08106=1200.416,187.035,-56.899,-177.792,6.361,148.503
C08107=1200.420,186.786,-56.876,-177.795,6.359,148.503
C08108=1200.424,186.537,-56.853,-177.798,6.358,148.504
C08109=1200.430,186.289,-56.830,-177.800,6.356,148.504
C08110=1200.434,186.040,-56.807,-177.803,6.354,148.504
C08111=1200.439,185.791,-56.784,-177.806,6.352,148.505
C08112=1200.443,185.542,-56.762,-177.808,6.350,148.505
C08113=1200.449,185.272,-56.736,-177.812,6.349,148.506
C08114=1200.453,185.003,-56.711,-177.814,6.347,148.506
C08115=1200.458,184.733,-56.686,-177.817,6.345,148.506
C08116=1200.463,184.464,-56.661,-177.820,6.343,148.507
C08117=1200.468,184.214,-56.639,-177.823,6.341,148.507
C08118=1200.473,183.966,-56.616,-177.825,6.340,148.507
C08119=1200.478,183.717,-56.593,-177.827,6.338,148.508
C08120=1200.482,183.468,-56.570,-177.830,6.336,148.508
C08121=1200.486,183.219,-56.547,-177.833,6.334,148.509
C08122=1200.491,182.970,-56.525,-177.835,6.333,148.509
C08123=1200.496,182.721,-56.502,-177.838,6.331,148.509
C08124=1200.501,182.472,-56.478,-177.841,6.329,148.510
C08125=1200.505,182.223,-56.456,-177.843,6.327,148.510
C08126=1200.510,181.974,-56.433,-177.846,6.325,148.510
C08127=1200.514,181.726,-56.411,-177.849,6.324,148.511
C08128=1200.519,181.476,-56.388,-177.851,6.322,148.511
C08129=1200.523,181.228,-56.365,-177.854,6.321,148.511
C08130=1200.528,180.979,-56.342,-177.856,6.319,148.512
C08131=1200.533,180.730,-56.320,-177.859,6.317,148.512
C08132=1200.537,180.481,-56.297,-177.862,6.316,148.513
C08133=1200.542,180.232,-56.273,-177.865,6.314,148.513
C08134=1200.547,179.983,-56.252,-177.867,6.312,148.513
C08135=1200.552,179.734,-56.228,-177.870,6.310,148.514
C08136=1200.556,179.486,-56.206,-177.873,6.309,148.514
C08137=1200.561,179.236,-56.183,-177.875,6.307,148.515
C08138=1200.565,178.988,-56.161,-177.878,6.305,148.515
C08139=1200.570,178.738,-56.138,-177.880,6.304,148.515
C08140=1200.574,178.489,-56.115,-177.883,6.302,148.516
C08141=1200.579,178.241,-56.093,-177.885,6.300,148.516
C08142=1200.584,177.992,-56.070,-177.888,6.299,148.516
C08143=1200.588,177.742,-56.048,-177.891,6.297,148.517
C08144=1200.593,177.494,-56.025,-177.893,6.295,148.517
C08145=1200.598,177.245,-56.003,-177.896,6.293,148.517
C08146=1200.602,176.996,-55.980,-177.899,6.291,148.518
C08147=1200.607,176.747,-55.958,-177.901,6.290,148.518
C08148=1200.612,176.498,-55.935,-177.904,6.289,148.519
C08149=1200.616,176.249,-55.913,-177.907,6.287,148.519
C08150=1200.621,176.001,-55.890,-177.909,6.285,148.519
C08151=1200.626,175.751,-55.867,-177.912,6.284,148.520
C08152=1200.630,175.502,-55.845,-177.915,6.282,148.520
C08153=1200.635,175.253,-55.822,-177.917,6.280,148.521
C08154=1200.640,175.004,-55.800,-177.919,6.279,148.521
C08155=1200.644,174.756,-55.778,-177.922,6.277,148.521
C08156=1200.649,174.506,-55.755,-177.925,6.275,148.522
C08157=1200.653,174.257,-55.733,-177.927,6.274,148.522
C08158=1200.658,174.009,-55.711,-177.930,6.272,148.522
C08159=1200.663,173.759,-55.688,-177.933,6.270,148.523
C08160=1200.667,173.510,-55.666,-177.935,6.268,148.523
C08161=1200.672,173.262,-55.644,-177.938,6.267,148.523
C08162=1200.677,173.012,-55.621,-177.941,6.266,148.524
C08163=1200.682,172.764,-55.600,-177.943,6.264,148.524
C08164=1200.686,172.515,-55.577,-177.946,6.262,148.525
C08165=1200.691,172.266,-55.554,-177.949,6.260,148.525
C08166=1200.696,172.017,-55.532,-177.951,6.258,148.526
C08167=1200.700,171.767,-55.510,-177.953,6.258,148.526
C08168=1200.704,171.519,-55.488,-177.956,6.256,148.526
C08169=1200.709,171.270,-55.465,-177.959,6.254,148.527
C08170=1200.714,171.021,-55.444,-177.961,6.252,148.527
C08171=1200.718,170.772,-55.422,-177.964,6.250,148.527
C08172=1200.723,170.524,-55.399,-177.967,6.249,148.528
C08173=1200.728,170.274,-55.377,-177.969,6.248,148.528
C08174=1200.733,170.025,-55.355,-177.972,6.246,148.529
C08175=1200.737,169.776,-55.333,-177.975,6.244,148.529
C08176=1200.742,169.527,-55.311,-177.977,6.242,148.529
C08177=1200.747,169.278,-55.288,-177.980,6.241,148.530
C08178=1200.752,169.029,-55.267,-177.983,6.239,148.530
C08179=1200.756,168.780,-55.244,-177.985,6.238,148.531
C08180=1200.761,168.532,-55.222,-177.987,6.236,148.531
C08181=1200.765,168.282,-55.200,-177.991,6.235,148.531
C08182=1200.771,168.033,-55.178,-177.993,6.233,148.532
C08183=1200.775,167.784,-55.156,-177.996,6.231,148.532
C08184=1200.780,167.536,-55.134,-177.998,6.230,148.533
C08185=1200.784,167.286,-55.112,-178.001,6.228,148.533
C08186=1200.789,167.038,-55.091,-178.003,6.226,148.533
C08187=1200.793,166.788,-55.069,-178.006,6.225,148.534
C08188=1200.798,166.540,-55.047,-178.009,6.223,148.534
C08189=1200.803,166.290,-55.024,-178.011,6.222,148.535
C08190=1200.808,166.041,-55.003,-178.014,6.220,148.535
C08191=1200.812,165.792,-54.980,-178.017,6.219,148.535
C08192=1200.817,165.543,-54.959,-178.019,6.217,148.536
C08193=1200.821,165.294,-54.937,-178.022,6.215,148.536
C08194=1200.826,165.045,-54.915,-178.024,6.214,148.537
C08195=1200.830,164.796,-54.893,-178.027,6.212,148.537
C08196=1200.835,164.547,-54.871,-178.030,6.211,148.537
C08197=1200.840,164.299,-54.850,-178.033,6.209,148.538
C08198=1200.844,164.049,-54.828,-178.035,6.207,148.538
C08199=1200.849,163.801,-54.806,-178.037,6.206,148.539
C08200=1200.854,163.551,-54.784,-178.040,6.205,148.539
C08201=1200.858,163.303,-54.762,-178.043,6.203,148.539
C08202=1200.863,163.053,-54.740,-178.046,6.201,148.540
C08203=1200.868,162.805,-54.718,-178.048,6.200,148.540
C08204=1200.873,162.555,-54.697,-178.051,6.199,148.541
C08205=1200.878,162.306,-54.675,-178.053,6.197,148.541
C08206=1200.883,162.057,-54.653,-178.056,6.195,148.541
C08207=1200.887,161.808,-54.631,-178.059,6.193,148.542
C08208=1200.891,161.560,-54.610,-178.061,6.192,148.542
C08209=1200.896,161.311,-54.588,-178.064,6.191,148.543
C08210=1200.901,161.061,-54.567,-178.067,6.189,148.543
C08211=1200.905,160.812,-54.545,-178.069,6.187,148.544
C08212=1200.910,160.564,-54.524,-178.071,6.186,148.544
C08213=1200.915,160.314,-54.502,-178.074,6.184,148.544
C08214=1200.920,160.065,-54.481,-178.077,6.183,148.545
C08215=1200.925,159.816,-54.459,-178.080,6.181,148.545
C08216=1200.929,159.567,-54.437,-178.082,6.180,148.546
C08217=1200.934,159.298,-54.414,-178.085,6.178,148.546
C08218=1200.939,159.029,-54.390,-178.088,6.177,148.547
C08219=1200.944,158.760,-54.367,-178.091,6.175,148.547
C08220=1200.949,158.491,-54.344,-178.093,6.173,148.547
C08221=1200.954,158.242,-54.322,-178.096,6.172,148.548
C08222=1200.959,157.994,-54.301,-178.099,6.170,148.548
C08223=1200.963,157.744,-54.279,-178.102,6.168,148.549
C08224=1200.968,157.495,-54.258,-178.104,6.167,148.549
C08225=1200.973,157.246,-54.237,-178.106,6.166,148.549
C08226=1200.978,156.996,-54.215,-178.109,6.164,148.550
C08227=1200.982,156.748,-54.193,-178.112,6.162,148.550
C08228=1200.987,156.499,-54.172,-178.114,6.161,148.551
C08229=1200.992,156.250,-54.151,-178.117,6.160,148.551
C08230=1200.996,156.001,-54.129,-178.120,6.158,148.552
C08231=1201.001,155.752,-54.108,-178.122,6.157,148.552
C08232=1201.006,155.503,-54.086,-178.125,6.155,148.553
C08233=1201.010,155.253,-54.065,-178.128,6.154,148.553
C08234=1201.015,155.005,-54.044,-178.130,6.152,148.553
C08235=1201.020,154.755,-54.023,-178.132,6.151,148.554
C08236=1201.025,154.507,-54.001,-178.136,6.149,148.554
C08237=1201.029,154.257,-53.980,-178.138,6.148,148.555
C08238=1201.034,154.008,-53.959,-178.141,6.146,148.555
C08239=1201.039,153.759,-53.938,-178.143,6.145,148.555
C08240=1201.044,153.511,-53.916,-178.146,6.143,148.556
C08241=1201.049,153.261,-53.895,-178.149,6.142,148.556
C08242=1201.052,153.012,-53.874,-178.151,6.141,148.557
C08243=1201.057,152.763,-53.853,-178.154,6.139,148.557
C08244=1201.062,152.514,-53.831,-178.156,6.137,148.558
C08245=1201.068,152.265,-53.810,-178.159,6.135,148.558
C08246=1201.071,152.016,-53.788,-178.162,6.135,148.559
C08247=1201.076,151.767,-53.768,-178.164,6.133,148.559
C08248=1201.081,151.518,-53.747,-178.167,6.131,148.559
C08249=1201.086,151.269,-53.725,-178.169,6.130,148.560
C08250=1201.091,151.020,-53.705,-178.172,6.129,148.560
C08251=1201.095,150.771,-53.682,-178.175,6.127,148.561
C08252=1201.099,150.522,-53.662,-178.177,6.126,148.561
C08253=1201.105,150.272,-53.641,-178.180,6.124,148.561
C08254=1201.109,150.024,-53.619,-178.183,6.123,148.562
C08255=1201.114,149.775,-53.599,-178.185,6.122,148.562
C08256=1201.119,149.526,-53.578,-178.188,6.120,148.563
C08257=1201.123,149.276,-53.556,-178.190,6.118,148.563
C08258=1201.128,149.027,-53.536,-178.194,6.117,148.564
C08259=1201.133,148.778,-53.515,-178.196,6.116,148.564
C08260=1201.138,148.529,-53.494,-178.198,6.114,148.565
C08261=1201.142,148.280,-53.473,-178.201,6.112,148.565
C08262=1201.147,148.031,-53.452,-178.204,6.112,148.566
C08263=1201.152,147.782,-53.431,-178.206,6.110,148.566
C08264=1201.156,147.532,-53.410,-178.209,6.108,148.566
C08265=1201.161,147.284,-53.388,-178.211,6.107,148.567
C08266=1201.166,147.035,-53.368,-178.214,6.106,148.567
C08267=1201.171,146.785,-53.347,-178.217,6.104,148.568
C08268=1201.175,146.536,-53.327,-178.219,6.103,148.568
C08269=1201.181,146.287,-53.306,-178.222,6.101,148.569
C08270=1201.185,146.039,-53.285,-178.225,6.100,148.569
C08271=1201.190,145.790,-53.264,-178.227,6.099,148.570
C08272=1201.195,145.540,-53.243,-178.230,6.097,148.570
C08273=1201.199,145.291,-53.222,-178.232,6.095,148.570
C08274=1201.204,145.041,-53.201,-178.235,6.094,148.571
C08275=1201.208,144.792,-53.181,-178.238,6.093,148.571
C08276=1201.213,144.544,-53.159,-178.240,6.091,148.572
C08277=1201.218,144.295,-53.138,-178.243,6.090,148.572
C08278=1201.223,144.046,-53.118,-178.246,6.089,148.573
C08279=1201.227,143.797,-53.097,-178.248,6.087,148.573
C08280=1201.233,143.547,-53.076,-178.250,6.086,148.573
C08281=1201.237,143.298,-53.056,-178.254,6.084,148.574
C08282=1201.242,143.049,-53.035,-178.256,6.083,148.574
C08283=1201.247,142.800,-53.014,-178.258,6.082,148.575
C08284=1201.251,142.551,-52.994,-178.261,6.080,148.575
C08285=1201.256,142.302,-52.973,-178.264,6.079,148.576
C08286=1201.261,142.053,-52.953,-178.266,6.077,148.576
C08287=1201.266,141.804,-52.932,-178.269,6.076,148.577
C08288=1201.270,141.554,-52.911,-178.272,6.075,148.577
C08289=1201.275,141.305,-52.890,-178.274,6.073,148.578
C08290=1201.279,141.056,-52.870,-178.277,6.071,148.578
C08291=1201.284,140.807,-52.849,-178.280,6.071,148.579
C08292=1201.289,140.558,-52.828,-178.282,6.069,148.579
C08293=1201.293,140.309,-52.808,-178.285,6.067,148.579
C08294=1201.299,140.060,-52.787,-178.287,6.066,148.580
C08295=1201.303,139.811,-52.767,-178.290,6.065,148.580
C08296=1201.307,139.562,-52.746,-178.292,6.064,148.581
C08297=1201.313,139.312,-52.725,-178.295,6.062,148.581
C08298=1201.317,139.063,-52.705,-178.298,6.061,148.582
C08299=1201.322,138.814,-52.685,-178.300,6.060,148.582
C08300=1201.327,138.565,-52.664,-178.303,6.058,148.583
C08301=1201.332,138.316,-52.644,-178.306,6.057,148.583
C08302=1201.336,138.067,-52.624,-178.308,6.056,148.584
C08303=1201.342,137.818,-52.603,-178.311,6.054,148.584
C08304=1201.346,137.569,-52.583,-178.314,6.053,148.585
C08305=1201.350,137.320,-52.562,-178.316,6.051,148.585
C08306=1201.356,137.070,-52.542,-178.319,6.050,148.585
C08307=1201.360,136.821,-52.522,-178.321,6.049,148.586
C08308=1201.365,136.572,-52.501,-178.324,6.047,148.586
C08309=1201.369,136.324,-52.481,-178.326,6.046,148.587
C08310=1201.374,136.074,-52.460,-178.329,6.045,148.587
C08311=1201.379,135.825,-52.440,-178.332,6.043,148.588
C08312=1201.384,135.576,-52.420,-178.334,6.042,148.588
C08313=1201.389,135.326,-52.399,-178.337,6.040,148.589
C08314=1201.393,135.078,-52.379,-178.340,6.040,148.589
C08315=1201.398,134.828,-52.359,-178.342,6.038,148.590
C08316=1201.403,134.580,-52.339,-178.345,6.036,148.590
C08317=1201.408,134.330,-52.318,-178.348,6.036,148.591
C08318=1201.413,134.081,-52.298,-178.350,6.034,148.591
C08319=1201.417,133.832,-52.278,-178.352,6.033,148.591
C08320=1201.422,133.583,-52.257,-178.356,6.031,148.592
C08321=1201.427,133.314,-52.236,-178.358,6.030,148.592
C08322=1201.432,133.046,-52.214,-178.361,6.028,148.593
C08323=1201.438,132.777,-52.192,-178.364,6.027,148.593
C08324=1201.443,132.508,-52.171,-178.367,6.026,148.594
C08325=1201.448,132.259,-52.150,-178.369,6.024,148.594
C08326=1201.452,132.010,-52.130,-178.372,6.024,148.595
C08327=1201.457,131.761,-52.110,-178.375,6.022,148.595
C08328=1201.461,131.512,-52.090,-178.377,6.021,148.596
C08329=1201.466,131.262,-52.070,-178.380,6.019,148.596
C08330=1201.471,131.013,-52.050,-178.383,6.018,148.597
C08331=1201.476,130.765,-52.029,-178.385,6.017,148.597
C08332=1201.481,130.515,-52.010,-178.388,6.015,148.598
C08333=1201.486,130.266,-51.989,-178.390,6.014,148.598
C08334=1201.490,130.017,-51.970,-178.393,6.013,148.599
C08335=1201.495,129.768,-51.949,-178.395,6.012,148.599
C08336=1201.500,129.519,-51.930,-178.398,6.010,148.600
C08337=1201.504,129.270,-51.910,-178.401,6.008,148.600
C08338=1201.509,129.020,-51.890,-178.403,6.008,148.601
C08339=1201.514,128.771,-51.870,-178.406,6.006,148.601
C08340=1201.518,128.522,-51.850,-178.409,6.005,148.602
C08341=1201.523,128.273,-51.829,-178.411,6.004,148.602
C08342=1201.528,128.024,-51.810,-178.413,6.003,148.603
C08343=1201.533,127.775,-51.789,-178.417,6.001,148.603
C08344=1201.538,127.525,-51.770,-178.419,6.000,148.604
C08345=1201.543,127.275,-51.750,-178.421,5.999,148.604
C08346=1201.548,127.027,-51.730,-178.425,5.997,148.605
C08347=1201.553,126.778,-51.710,-178.427,5.996,148.605
C08348=1201.557,126.529,-51.690,-178.430,5.995,148.606
C08349=1201.562,126.279,-51.670,-178.432,5.994,148.606
C08350=1201.567,126.030,-51.651,-178.435,5.992,148.606
C08351=1201.572,125.781,-51.631,-178.437,5.991,148.607
C08352=1201.576,125.532,-51.611,-178.440,5.990,148.607
C08353=1201.581,125.282,-51.591,-178.443,5.989,148.608
C08354=1201.586,125.033,-51.571,-178.445,5.987,148.608
C08355=1201.591,124.784,-51.552,-178.447,5.986,148.609
C08356=1201.595,124.535,-51.533,-178.451,5.985,148.609
C08357=1201.599,124.286,-51.512,-178.453,5.984,148.610
C08358=1201.605,124.037,-51.493,-178.455,5.982,148.610
C08359=1201.609,123.788,-51.473,-178.458,5.982,148.611
C08360=1201.614,123.539,-51.453,-178.461,5.980,148.611
C08361=1201.619,123.289,-51.433,-178.464,5.978,148.612
C08362=1201.624,123.040,-51.414,-178.466,5.977,148.612
C08363=1201.629,122.791,-51.394,-178.469,5.976,148.613
C08364=1201.633,122.542,-51.374,-178.471,5.975,148.613
C08365=1201.638,122.293,-51.355,-178.474,5.973,148.614
C08366=1201.643,122.043,-51.335,-178.477,5.973,148.614
C08367=1201.648,121.794,-51.315,-178.479,5.971,148.615
C08368=1201.653,121.545,-51.297,-178.481,5.970,148.615
C08369=1201.657,121.296,-51.276,-178.485,5.969,148.616
C08370=1201.662,121.047,-51.257,-178.487,5.968,148.616
C08371=1201.667,120.798,-51.237,-178.490,5.966,148.617
C08372=1201.672,120.548,-51.218,-178.492,5.965,148.617
C08373=1201.677,120.299,-51.198,-178.495,5.964,148.618
C08374=1201.682,120.050,-51.179,-178.497,5.963,148.618
C08375=1201.686,119.801,-51.159,-178.500,5.961,148.619
C08376=1201.690,119.552,-51.139,-178.503,5.961,148.619
C08377=1201.696,119.303,-51.120,-178.505,5.959,148.620
C08378=1201.700,119.053,-51.100,-178.508,5.958,148.620
C08379=1201.705,118.804,-51.081,-178.511,5.956,148.621
C08380=1201.710,118.555,-51.061,-178.513,5.956,148.621
C08381=1201.715,118.306,-51.042,-178.516,5.954,148.622
C08382=1201.720,118.057,-51.023,-178.518,5.953,148.622
C08383=1201.725,117.807,-51.003,-178.521,5.952,148.623
C08384=1201.729,117.558,-50.984,-178.523,5.951,148.623
C08385=1201.734,117.309,-50.965,-178.527,5.949,148.624
C08386=1201.739,117.059,-50.945,-178.529,5.948,148.624
C08387=1201.744,116.811,-50.926,-178.531,5.947,148.625
C08388=1201.749,116.561,-50.906,-178.534,5.946,148.625
C08389=1201.753,116.312,-50.887,-178.537,5.944,148.626
C08390=1201.758,116.063,-50.868,-178.539,5.944,148.626
C08391=1201.763,115.813,-50.848,-178.541,5.943,148.627
C08392=1201.768,115.564,-50.829,-178.545,5.941,148.627
C08393=1201.772,115.315,-50.810,-178.547,5.940,148.628
C08394=1201.777,115.066,-50.790,-178.550,5.939,148.628
C08395=1201.782,114.817,-50.771,-178.552,5.938,148.629
C08396=1201.786,114.567,-50.752,-178.555,5.936,148.629
C08397=1201.792,114.319,-50.733,-178.557,5.936,148.630
C08398=1201.796,114.069,-50.713,-178.560,5.934,148.630
C08399=1201.802,113.820,-50.694,-178.563,5.933,148.631
C08400=1201.806,113.571,-50.675,-178.565,5.932,148.631
C08401=1201.811,113.321,-50.656,-178.568,5.931,148.632
C08402=1201.816,113.072,-50.636,-178.571,5.929,148.632
C08403=1201.821,112.823,-50.618,-178.573,5.929,148.633
C08404=1201.825,112.574,-50.598,-178.576,5.927,148.633
C08405=1201.830,112.325,-50.579,-178.579,5.926,148.634
C08406=1201.835,112.076,-50.560,-178.581,5.925,148.634
C08407=1201.840,111.826,-50.541,-178.583,5.924,148.635
C08408=1201.844,111.577,-50.522,-178.586,5.923,148.635
C08409=1201.850,111.328,-50.503,-178.589,5.921,148.636
C08410=1201.855,111.078,-50.483,-178.591,5.921,148.637
C08411=1201.859,110.830,-50.464,-178.594,5.919,148.637
C08412=1201.864,110.580,-50.446,-178.597,5.918,148.638
C08413=1201.869,110.331,-50.427,-178.599,5.917,148.638
C08414=1201.874,110.082,-50.407,-178.602,5.916,148.639
C08415=1201.878,109.833,-50.388,-178.604,5.915,148.639
C08416=1201.883,109.583,-50.370,-178.607,5.914,148.640
C08417=1201.889,109.334,-50.350,-178.609,5.913,148.640
C08418=1201.893,109.085,-50.331,-178.613,5.911,148.641
C08419=1201.898,108.835,-50.313,-178.615,5.910,148.641
C08420=1201.902,108.586,-50.294,-178.618,5.909,148.642
C08421=1201.908,108.337,-50.274,-178.620,5.908,148.642
C08422=1201.912,108.088,-50.255,-178.623,5.907,148.643
C08423=1201.917,107.838,-50.237,-178.625,5.906,148.643
C08424=1201.921,107.589,-50.218,-178.628,5.905,148.644
C08425=1201.927,107.320,-50.198,-178.631,5.903,148.644
C08426=1201.933,107.053,-50.177,-178.634,5.902,148.645
C08427=1201.937,106.784,-50.157,-178.636,5.901,148.646
C08428=1201.943,106.516,-50.136,-178.639,5.900,148.646
C08429=1201.947,106.266,-50.117,-178.642,5.899,148.647
C08430=1201.952,106.017,-50.099,-178.644,5.897,148.647
C08431=1201.957,105.768,-50.080,-178.647,5.897,148.648
C08432=1201.962,105.518,-50.061,-178.649,5.896,148.648
C08433=1201.966,105.270,-50.042,-178.652,5.894,148.649
C08434=1201.972,105.019,-50.023,-178.654,5.893,148.649
C08435=1201.976,104.771,-50.005,-178.658,5.892,148.650
C08436=1201.982,104.521,-49.986,-178.660,5.891,148.650
C08437=1201.986,104.272,-49.967,-178.662,5.890,148.651
C08438=1201.990,104.024,-49.948,-178.665,5.889,148.651
C08439=1201.996,103.774,-49.930,-178.668,5.888,148.652
C08440=1202.000,103.525,-49.911,-178.670,5.886,148.652
C08441=1202.006,103.275,-49.892,-178.673,5.886,148.653
C08442=1202.010,103.025,-49.874,-178.675,5.885,148.653
C08443=1202.015,102.777,-49.855,-178.678,5.883,148.654
C08444=1202.020,102.527,-49.837,-178.680,5.883,148.654
C08445=1202.024,102.278,-49.818,-178.684,5.881,148.655
C08446=1202.029,102.029,-49.800,-178.686,5.880,148.655
C08447=1202.035,101.780,-49.780,-178.688,5.880,148.656
C08448=1202.039,101.530,-49.762,-178.691,5.878,148.656
C08449=1202.043,101.282,-49.743,-178.694,5.877,148.657
C08450=1202.049,101.032,-49.725,-178.696,5.876,148.657
C08451=1202.053,100.782,-49.706,-178.699,5.875,148.658
C08452=1202.058,100.534,-49.688,-178.701,5.874,148.659
C08453=1202.064,100.284,-49.669,-178.704,5.873,148.659
C08454=1202.068,100.035,-49.650,-178.706,5.872,148.660
C08455=1202.073,99.786,-49.632,-178.709,5.871,148.660
C08456=1202.078,99.536,-49.613,-178.712,5.869,148.661
C08457=1202.083,99.288,-49.595,-178.714,5.869,148.661
C08458=1202.087,99.038,-49.576,-178.718,5.867,148.662
C08459=1202.093,98.788,-49.558,-178.720,5.866,148.662
C08460=1202.098,98.539,-49.540,-178.722,5.866,148.663
C08461=1202.102,98.290,-49.521,-178.725,5.864,148.663
C08462=1202.107,98.041,-49.503,-178.728,5.864,148.664
C08463=1202.112,97.791,-49.484,-178.730,5.863,148.664
C08464=1202.117,97.543,-49.465,-178.733,5.861,148.665
C08465=1202.121,97.293,-49.447,-178.735,5.860,148.666
C08466=1202.126,97.044,-49.429,-178.738,5.859,148.666
C08467=1202.131,96.795,-49.411,-178.740,5.858,148.667
C08468=1202.136,96.545,-49.392,-178.743,5.857,148.667
C08469=1202.141,96.296,-49.374,-178.746,5.856,148.668
C08470=1202.146,96.047,-49.356,-178.748,5.855,148.668
C08471=1202.151,95.797,-49.338,-178.751,5.854,148.669
C08472=1202.156,95.548,-49.319,-178.754,5.853,148.669
C08473=1202.160,95.299,-49.300,-178.756,5.852,148.670
C08474=1202.165,95.050,-49.282,-178.758,5.851,148.670
C08475=1202.170,94.800,-49.264,-178.762,5.850,148.671
C08476=1202.175,94.551,-49.246,-178.764,5.849,148.672
C08477=1202.179,94.301,-49.228,-178.766,5.848,148.672
C08478=1202.185,94.052,-49.209,-178.769,5.847,148.673
C08479=1202.189,93.803,-49.190,-178.772,5.846,148.673
C08480=1202.194,93.554,-49.172,-178.774,5.845,148.674
C08481=1202.199,93.305,-49.154,-178.777,5.844,148.674
C08482=1202.204,93.055,-49.136,-178.780,5.843,148.675
C08483=1202.209,92.806,-49.118,-178.782,5.842,148.675
C08484=1202.213,92.557,-49.100,-178.785,5.841,148.676
C08485=1202.218,92.308,-49.082,-178.787,5.840,148.676
C08486=1202.224,92.058,-49.064,-178.790,5.839,148.677
C08487=1202.228,91.808,-49.045,-178.792,5.838,148.677
C08488=1202.233,91.559,-49.027,-178.795,5.837,148.678
C08489=1202.238,91.310,-49.009,-178.797,5.836,148.679
C08490=1202.243,91.061,-48.991,-178.800,5.835,148.679
C08491=1202.248,90.811,-48.973,-178.803,5.834,148.680
C08492=1202.253,90.562,-48.955,-178.805,5.833,148.680
C08493=1202.257,90.312,-48.937,-178.808,5.832,148.681
C08494=1202.262,90.063,-48.919,-178.811,5.831,148.681
C08495=1202.267,89.814,-48.901,-178.813,5.830,148.682
C08496=1202.272,89.565,-48.883,-178.816,5.829,148.682
C08497=1202.277,89.316,-48.865,-178.818,5.828,148.683
C08498=1202.282,89.067,-48.847,-178.821,5.827,148.684
C08499=1202.287,88.817,-48.829,-178.824,5.826,148.684
C08500=1202.292,88.568,-48.811,-178.826,5.825,148.685
C08501=1202.296,88.318,-48.793,-178.829,5.824,148.685
C08502=1202.301,88.069,-48.775,-178.832,5.823,148.686
C08503=1202.306,87.820,-48.757,-178.834,5.822,148.686
C08504=1202.311,87.571,-48.739,-178.837,5.821,148.687
C08505=1202.316,87.322,-48.721,-178.839,5.821,148.688
C08506=1202.320,87.072,-48.703,-178.842,5.819,148.688
C08507=1202.326,86.823,-48.686,-178.844,5.818,148.689
C08508=1202.331,86.573,-48.668,-178.847,5.817,148.689
C08509=1202.335,86.324,-48.650,-178.850,5.816,148.690
C08510=1202.340,86.075,-48.632,-178.852,5.816,148.690
C08511=1202.345,85.825,-48.613,-178.855,5.815,148.691
C08512=1202.350,85.576,-48.595,-178.858,5.813,148.691
C08513=1202.355,85.326,-48.578,-178.860,5.812,148.692
C08514=1202.360,85.077,-48.560,-178.863,5.812,148.693
C08515=1202.365,84.828,-48.542,-178.865,5.811,148.693
C08516=1202.370,84.579,-48.524,-178.868,5.809,148.694
C08517=1202.374,84.330,-48.507,-178.870,5.809,148.694
C08518=1202.379,84.080,-48.490,-178.873,5.808,148.695
C08519=1202.384,83.831,-48.472,-178.876,5.807,148.695
C08520=1202.389,83.582,-48.454,-178.878,5.806,148.696
C08521=1202.394,83.333,-48.436,-178.881,5.805,148.696
C08522=1202.399,83.083,-48.418,-178.883,5.804,148.697
C08523=1202.404,82.834,-48.400,-178.886,5.803,148.697
C08524=1202.409,82.584,-48.382,-178.889,5.802,148.698
C08525=1202.413,82.335,-48.366,-178.891,5.802,148.699
C08526=1202.418,82.086,-48.348,-178.894,5.800,148.699
C08527=1202.423,81.837,-48.330,-178.896,5.799,148.700
C08528=1202.428,81.587,-48.312,-178.899,5.798,148.700
C08529=1202.433,81.318,-48.293,-178.902,5.797,148.701
C08530=1202.438,81.050,-48.274,-178.904,5.796,148.702
C08531=1202.444,80.781,-48.255,-178.907,5.796,148.702
C08532=1202.449,80.514,-48.236,-178.910,5.794,148.703
C08533=1202.454,80.264,-48.219,-178.912,5.794,148.703
C08534=1202.459,80.015,-48.201,-178.915,5.793,148.704
C08535=1202.464,79.766,-48.183,-178.918,5.792,148.705
C08536=1202.469,79.516,-48.166,-178.920,5.791,148.705
C08537=1202.474,79.267,-48.148,-178.923,5.790,148.706
C08538=1202.478,79.018,-48.131,-178.925,5.789,148.706
C08539=1202.483,78.768,-48.113,-178.928,5.788,148.707
C08540=1202.489,78.519,-48.096,-178.931,5.787,148.707
C08541=1202.493,78.269,-48.078,-178.933,5.786,148.708
C08542=1202.498,78.021,-48.061,-178.936,5.786,148.709
C08543=1202.503,77.771,-48.043,-178.939,5.784,148.709
C08544=1202.508,77.522,-48.025,-178.941,5.784,148.710
C08545=1202.513,77.272,-48.008,-178.944,5.783,148.710
C08546=1202.517,77.023,-47.991,-178.946,5.782,148.711
C08547=1202.522,76.773,-47.974,-178.949,5.781,148.711
C08548=1202.527,76.524,-47.956,-178.952,5.780,148.712
C08549=1202.532,76.274,-47.939,-178.954,5.779,148.712
C08550=1202.537,76.025,-47.921,-178.956,5.779,148.713
C08551=1202.542,75.776,-47.904,-178.960,5.777,148.714
C08552=1202.547,75.527,-47.887,-178.962,5.776,148.714
C08553=1202.552,75.277,-47.869,-178.964,5.776,148.715
C08554=1202.557,75.028,-47.852,-178.967,5.775,148.715
C08555=1202.561,74.779,-47.835,-178.970,5.773,148.716
C08556=1202.566,74.529,-47.817,-178.972,5.773,148.717
C08557=1202.571,74.280,-47.800,-178.975,5.772,148.717
C08558=1202.576,74.030,-47.783,-178.977,5.771,148.718
C08559=1202.581,73.781,-47.766,-178.980,5.771,148.718
C08560=1202.587,73.532,-47.748,-178.982,5.769,148.719
C08561=1202.591,73.283,-47.731,-178.985,5.769,148.719
C08562=1202.596,73.033,-47.713,-178.988,5.768,148.720
C08563=1202.600,72.784,-47.697,-178.990,5.767,148.720
C08564=1202.606,72.534,-47.679,-178.993,5.766,148.721
C08565=1202.611,72.285,-47.661,-178.996,5.765,148.722
C08566=1202.615,72.036,-47.645,-178.998,5.764,148.722
C08567=1202.621,71.786,-47.628,-179.000,5.764,148.723
C08568=1202.625,71.538,-47.610,-179.003,5.763,148.724
C08569=1202.630,71.288,-47.593,-179.006,5.761,148.724
C08570=1202.636,71.038,-47.576,-179.008,5.761,148.725
C08571=1202.640,70.788,-47.559,-179.011,5.760,148.725
C08572=1202.645,70.539,-47.541,-179.013,5.759,148.726
C08573=1202.650,70.291,-47.525,-179.016,5.758,148.726
C08574=1202.655,70.041,-47.508,-179.019,5.757,148.727
C08575=1202.660,69.791,-47.491,-179.021,5.757,148.727
C08576=1202.665,69.542,-47.473,-179.024,5.756,148.728
C08577=1202.669,69.293,-47.456,-179.026,5.755,148.729
C08578=1202.674,69.043,-47.439,-179.029,5.754,148.729
C08579=1202.679,68.794,-47.423,-179.032,5.753,148.730
C08580=1202.684,68.545,-47.405,-179.034,5.752,148.730
C08581=1202.689,68.295,-47.388,-179.037,5.752,148.731
C08582=1202.694,68.046,-47.371,-179.039,5.751,148.732
C08583=1202.699,67.797,-47.355,-179.042,5.749,148.732
C08584=1202.704,67.547,-47.337,-179.045,5.749,148.733
C08585=1202.709,67.297,-47.321,-179.047,5.748,148.733
C08586=1202.714,67.048,-47.303,-179.049,5.747,148.734
C08587=1202.718,66.799,-47.286,-179.052,5.747,148.734
C08588=1202.724,66.550,-47.269,-179.055,5.746,148.735
C08589=1202.728,66.300,-47.252,-179.057,5.745,148.736
C08590=1202.733,66.051,-47.236,-179.060,5.744,148.736
C08591=1202.738,65.801,-47.219,-179.063,5.743,148.737
C08592=1202.743,65.552,-47.202,-179.065,5.743,148.738
C08593=1202.748,65.302,-47.185,-179.067,5.742,148.738
C08594=1202.753,65.053,-47.168,-179.071,5.741,148.739
C08595=1202.758,64.804,-47.150,-179.073,5.740,148.739
C08596=1202.763,64.555,-47.134,-179.075,5.739,148.740
C08597=1202.767,64.305,-47.117,-179.078,5.739,148.740
C08598=1202.773,64.056,-47.100,-179.081,5.738,148.741
C08599=1202.778,63.807,-47.084,-179.083,5.737,148.741
C08600=1202.783,63.557,-47.066,-179.086,5.736,148.742
C08601=1202.787,63.308,-47.050,-179.089,5.735,148.743
C08602=1202.792,63.058,-47.033,-179.091,5.734,148.743
C08603=1202.798,62.809,-47.016,-179.093,5.734,148.744
C08604=1202.802,62.560,-47.000,-179.096,5.733,148.745
C08605=1202.807,62.310,-46.983,-179.098,5.732,148.745
C08606=1202.812,62.061,-46.966,-179.101,5.731,148.746
C08607=1202.817,61.811,-46.949,-179.104,5.730,148.746
C08608=1202.821,61.562,-46.933,-179.106,5.730,148.747
C08609=1202.827,61.313,-46.916,-179.109,5.729,148.747
C08610=1202.832,61.063,-46.900,-179.111,5.728,148.748
C08611=1202.837,60.813,-46.883,-179.114,5.728,148.749
C08612=1202.842,60.564,-46.866,-179.117,5.726,148.749
C08613=1202.847,60.315,-46.850,-179.119,5.726,148.750
C08614=1202.851,60.065,-46.833,-179.122,5.725,148.751
C08615=1202.856,59.816,-46.817,-179.124,5.724,148.751
C08616=1202.862,59.567,-46.799,-179.127,5.724,148.752
C08617=1202.866,59.317,-46.783,-179.129,5.723,148.752
C08618=1202.871,59.068,-46.766,-179.132,5.722,148.753
C08619=1202.877,58.818,-46.750,-179.135,5.721,148.753
C08620=1202.881,58.569,-46.733,-179.137,5.720,148.754
C08621=1202.886,58.320,-46.717,-179.140,5.720,148.755
C08622=1202.891,58.070,-46.700,-179.142,5.719,148.755
C08623=1202.897,57.821,-46.683,-179.145,5.718,148.756
C08624=1202.901,57.572,-46.667,-179.147,5.718,148.756
C08625=1202.906,57.322,-46.651,-179.150,5.717,148.757
C08626=1202.911,57.073,-46.634,-179.153,5.715,148.758
C08627=1202.915,56.823,-46.618,-179.155,5.715,148.758
C08628=1202.921,56.574,-46.601,-179.158,5.714,148.759
C08629=1202.926,56.325,-46.584,-179.160,5.713,148.759
C08630=1202.930,56.075,-46.568,-179.163,5.713,148.760
C08631=1202.936,55.826,-46.552,-179.166,5.712,148.761
C08632=1202.940,55.576,-46.535,-179.168,5.711,148.761
C08633=1202.946,55.308,-46.518,-179.171,5.710,148.762
C08634=1202.951,55.039,-46.499,-179.174,5.710,148.762
C08635=1202.957,54.771,-46.482,-179.176,5.709,148.763
C08636=1202.962,54.503,-46.465,-179.179,5.708,148.764
C08637=1202.966,54.253,-46.448,-179.182,5.707,148.764
C08638=1202.972,54.003,-46.432,-179.184,5.706,148.765
C08639=1202.977,53.754,-46.415,-179.187,5.706,148.766
C08640=1202.981,53.504,-46.399,-179.189,5.705,148.766
C08641=1202.987,53.255,-46.383,-179.192,5.705,148.767
C08642=1202.991,53.006,-46.366,-179.194,5.704,148.767
C08643=1202.996,52.757,-46.350,-179.197,5.703,148.768
C08644=1203.001,52.507,-46.334,-179.199,5.703,148.769
C08645=1203.006,52.258,-46.318,-179.203,5.701,148.769
C08646=1203.012,52.008,-46.301,-179.205,5.700,148.770
C08647=1203.017,51.759,-46.285,-179.207,5.700,148.770
C08648=1203.021,51.509,-46.268,-179.210,5.699,148.771
C08649=1203.027,51.260,-46.253,-179.212,5.698,148.772
C08650=1203.031,51.010,-46.236,-179.215,5.698,148.772
C08651=1203.036,50.761,-46.220,-179.218,5.697,148.773
C08652=1203.041,50.511,-46.204,-179.220,5.697,148.774
C08653=1203.046,50.263,-46.187,-179.222,5.696,148.774
C08654=1203.051,50.013,-46.171,-179.225,5.695,148.775
C08655=1203.056,49.764,-46.155,-179.228,5.694,148.775
C08656=1203.061,49.514,-46.139,-179.231,5.693,148.776
C08657=1203.066,49.265,-46.123,-179.233,5.693,148.776
C08658=1203.071,49.015,-46.107,-179.236,5.692,148.777
C08659=1203.076,48.766,-46.091,-179.238,5.691,148.778
C08660=1203.080,48.516,-46.075,-179.241,5.691,148.778
C08661=1203.086,48.267,-46.058,-179.243,5.690,148.779
C08662=1203.090,48.017,-46.042,-179.246,5.689,148.780
C08663=1203.095,47.768,-46.026,-179.248,5.689,148.780
C08664=1203.100,47.518,-46.010,-179.251,5.688,148.781
C08665=1203.106,47.269,-45.995,-179.253,5.688,148.781
C08666=1203.110,47.019,-45.978,-179.256,5.686,148.782
C08667=1203.115,46.770,-45.962,-179.259,5.686,148.783
C08668=1203.120,46.521,-45.946,-179.261,5.685,148.783
C08669=1203.125,46.271,-45.930,-179.264,5.684,148.784
C08670=1203.130,46.022,-45.914,-179.266,5.684,148.784
C08671=1203.135,45.772,-45.898,-179.269,5.683,148.785
C08672=1203.141,45.523,-45.882,-179.271,5.682,148.786
C08673=1203.145,45.273,-45.866,-179.274,5.682,148.786
C08674=1203.150,45.024,-45.850,-179.276,5.681,148.787
C08675=1203.155,44.775,-45.834,-179.279,5.681,148.788
C08676=1203.160,44.525,-45.818,-179.281,5.680,148.788
C08677=1203.165,44.276,-45.803,-179.284,5.679,148.789
C08678=1203.169,44.026,-45.786,-179.286,5.679,148.789
C08679=1203.175,43.777,-45.770,-179.289,5.678,148.790
C08680=1203.180,43.528,-45.755,-179.292,5.676,148.790
C08681=1203.185,43.278,-45.738,-179.294,5.676,148.791
C08682=1203.190,43.029,-45.723,-179.297,5.675,148.792
C08683=1203.195,42.779,-45.707,-179.300,5.675,148.792
C08684=1203.200,42.529,-45.691,-179.302,5.674,148.793
C08685=1203.205,42.281,-45.675,-179.305,5.673,148.794
C08686=1203.209,42.031,-45.659,-179.307,5.673,148.794
C08687=1203.215,41.781,-45.644,-179.310,5.672,148.795
C08688=1203.220,41.532,-45.628,-179.312,5.672,148.796
C08689=1203.225,41.282,-45.612,-179.315,5.671,148.796
C08690=1203.230,41.033,-45.596,-179.317,5.670,148.797
C08691=1203.235,40.784,-45.581,-179.320,5.670,148.797
C08692=1203.239,40.534,-45.565,-179.323,5.669,148.798
C08693=1203.245,40.285,-45.549,-179.325,5.668,148.799
C08694=1203.250,40.036,-45.533,-179.327,5.668,148.799
C08695=1203.255,39.785,-45.517,-179.330,5.667,148.800
C08696=1203.260,39.536,-45.502,-179.333,5.667,148.801
C08697=1203.265,39.287,-45.487,-179.335,5.666,148.801
C08698=1203.269,39.037,-45.470,-179.337,5.665,148.802
C08699=1203.275,38.788,-45.454,-179.340,5.665,148.802
C08700=1203.280,38.539,-45.439,-179.343,5.664,148.803
C08701=1203.284,38.289,-45.423,-179.345,5.663,148.803
C08702=1203.289,38.039,-45.408,-179.348,5.662,148.804
C08703=1203.295,37.790,-45.392,-179.351,5.662,148.805
C08704=1203.300,37.540,-45.376,-179.353,5.661,148.805
C08705=1203.304,37.291,-45.361,-179.356,5.661,148.806
C08706=1203.309,37.042,-45.345,-179.358,5.660,148.807
C08707=1203.315,36.793,-45.329,-179.361,5.659,148.807
C08708=1203.319,36.543,-45.313,-179.363,5.659,148.808
C08709=1203.324,36.293,-45.298,-179.366,5.658,148.809
C08710=1203.330,36.044,-45.283,-179.368,5.657,148.809
C08711=1203.334,35.794,-45.267,-179.371,5.657,148.810
C08712=1203.339,35.545,-45.252,-179.374,5.656,148.810
C08713=1203.344,35.295,-45.236,-179.376,5.656,148.811
C08714=1203.350,35.046,-45.221,-179.379,5.655,148.812
C08715=1203.355,34.796,-45.205,-179.381,5.654,148.812
C08716=1203.359,34.547,-45.190,-179.384,5.654,148.813
C08717=1203.365,34.297,-45.174,-179.386,5.653,148.814
C08718=1203.370,34.048,-45.159,-179.389,5.653,148.814
C08719=1203.374,33.798,-45.143,-179.391,5.652,148.815
C08720=1203.379,33.549,-45.128,-179.394,5.651,148.815
C08721=1203.385,33.299,-45.112,-179.396,5.651,148.816
C08722=1203.389,33.050,-45.097,-179.399,5.650,148.817
C08723=1203.395,32.801,-45.081,-179.402,5.650,148.817
C08724=1203.399,32.551,-45.066,-179.404,5.649,148.818
C08725=1203.404,32.302,-45.051,-179.406,5.648,148.819
C08726=1203.410,32.052,-45.035,-179.409,5.648,148.819
C08727=1203.414,31.803,-45.020,-179.412,5.647,148.820
C08728=1203.419,31.553,-45.004,-179.414,5.647,148.821
C08729=1203.424,31.303,-44.990,-179.416,5.646,148.821
C08730=1203.429,31.054,-44.974,-179.419,5.645,148.822
C08731=1203.435,30.805,-44.959,-179.422,5.645,148.822
C08732=1203.439,30.556,-44.944,-179.424,5.644,148.823
C08733=1203.444,30.305,-44.928,-179.427,5.643,148.823
C08734=1203.449,30.056,-44.913,-179.429,5.643,148.824
C08735=1203.454,29.807,-44.897,-179.432,5.642,148.825
C08736=1203.459,29.558,-44.882,-179.435,5.642,148.826
C08737=1203.465,29.289,-44.866,-179.437,5.641,148.826
C08738=1203.470,29.020,-44.849,-179.440,5.641,148.827
C08739=1203.475,28.752,-44.833,-179.442,5.640,148.828
C08740=1203.481,28.482,-44.817,-179.446,5.639,148.828
C08741=1203.486,28.233,-44.802,-179.448,5.638,148.829
C08742=1203.491,27.983,-44.786,-179.451,5.638,148.830
C08743=1203.495,27.734,-44.771,-179.453,5.637,148.830
C08744=1203.501,27.485,-44.755,-179.456,5.636,148.831
C08745=1203.506,27.235,-44.741,-179.458,5.636,148.831
C08746=1203.511,26.986,-44.725,-179.461,5.635,148.832
C08747=1203.516,26.737,-44.710,-179.463,5.634,148.833
C08748=1203.521,26.487,-44.695,-179.465,5.635,148.833
C08749=1203.526,26.237,-44.680,-179.468,5.634,148.834
C08750=1203.531,25.987,-44.664,-179.471,5.634,148.835
C08751=1203.536,25.738,-44.650,-179.473,5.633,148.835
C08752=1203.541,25.488,-44.635,-179.476,5.633,148.836
C08753=1203.546,25.239,-44.620,-179.478,5.632,148.836
C08754=1203.551,24.990,-44.604,-179.481,5.631,148.837
C08755=1203.556,24.741,-44.589,-179.483,5.631,148.838
C08756=1203.562,24.491,-44.574,-179.486,5.630,148.838
C08757=1203.566,24.241,-44.559,-179.489,5.630,148.839
C08758=1203.571,23.992,-44.544,-179.491,5.629,148.840
C08759=1203.576,23.742,-44.529,-179.493,5.628,148.840
C08760=1203.581,23.493,-44.514,-179.496,5.628,148.841
C08761=1203.586,23.243,-44.498,-179.499,5.627,148.842
C08762=1203.591,22.993,-44.484,-179.501,5.627,148.842
C08763=1203.596,22.744,-44.469,-179.504,5.626,148.843
C08764=1203.601,22.494,-44.454,-179.506,5.625,148.843
C08765=1203.606,22.245,-44.439,-179.509,5.625,148.844
C08766=1203.611,21.996,-44.424,-179.511,5.624,148.845
C08767=1203.616,21.746,-44.409,-179.514,5.624,148.845
C08768=1203.621,21.497,-44.394,-179.516,5.623,148.846
C08769=1203.627,21.247,-44.380,-179.519,5.622,148.847
C08770=1203.631,20.998,-44.365,-179.522,5.622,148.847
C08771=1203.636,20.748,-44.350,-179.524,5.621,148.848
C08772=1203.642,20.499,-44.335,-179.527,5.621,148.849
C08773=1203.647,20.249,-44.320,-179.529,5.620,148.849
C08774=1203.651,20.000,-44.305,-179.532,5.620,148.850
C08775=1203.657,19.751,-44.290,-179.534,5.620,148.850
C08776=1203.662,19.501,-44.276,-179.536,5.619,148.851
C08777=1203.666,19.252,-44.261,-179.539,5.619,148.852
C08778=1203.672,19.002,-44.246,-179.542,5.618,148.852
C08779=1203.677,18.753,-44.231,-179.544,5.617,148.853
C08780=1203.682,18.503,-44.216,-179.546,5.617,148.854
C08781=1203.687,18.253,-44.202,-179.549,5.616,148.854
C08782=1203.692,18.004,-44.187,-179.552,5.616,148.855
C08783=1203.697,17.754,-44.172,-179.554,5.615,148.856
C08784=1203.701,17.505,-44.157,-179.557,5.615,148.856
C08785=1203.707,17.255,-44.142,-179.559,5.614,148.857
C08786=1203.712,17.006,-44.127,-179.562,5.613,148.857
C08787=1203.717,16.756,-44.113,-179.565,5.613,148.858
C08788=1203.721,16.507,-44.098,-179.567,5.612,148.859
C08789=1203.727,16.257,-44.083,-179.570,5.612,148.860
C08790=1203.732,16.007,-44.069,-179.571,5.612,148.860
C08791=1203.737,15.758,-44.054,-179.574,5.611,148.861
C08792=1203.742,15.509,-44.040,-179.577,5.611,148.861
C08793=1203.747,15.259,-44.025,-179.579,5.610,148.862
C08794=1203.752,15.010,-44.010,-179.582,5.610,148.863
C08795=1203.757,14.760,-43.996,-179.585,5.609,148.863
C08796=1203.762,14.511,-43.981,-179.587,5.608,148.864
C08797=1203.767,14.261,-43.966,-179.589,5.608,148.865
C08798=1203.772,14.011,-43.951,-179.592,5.607,148.865
C08799=1203.777,13.761,-43.937,-179.595,5.607,148.866
C08800=1203.782,13.512,-43.922,-179.597,5.606,148.867
C08801=1203.787,13.262,-43.908,-179.600,5.606,148.867
C08802=1203.792,13.013,-43.894,-179.602,5.605,148.868
C08803=1203.797,12.763,-43.878,-179.604,5.605,148.868
C08804=1203.803,12.514,-43.864,-179.607,5.605,148.869
C08805=1203.808,12.265,-43.850,-179.610,5.604,148.870
C08806=1203.812,12.016,-43.835,-179.612,5.604,148.870
C08807=1203.817,11.766,-43.821,-179.615,5.603,148.871
C08808=1203.822,11.516,-43.806,-179.617,5.602,148.872
C08809=1203.827,11.266,-43.792,-179.620,5.602,148.872
C08810=1203.833,11.016,-43.777,-179.622,5.601,148.873
C08811=1203.838,10.767,-43.762,-179.625,5.601,148.874
C08812=1203.843,10.518,-43.748,-179.628,5.600,148.874
C08813=1203.847,10.268,-43.734,-179.630,5.600,148.875
C08814=1203.853,10.019,-43.720,-179.632,5.600,148.875
C08815=1203.858,9.770,-43.705,-179.635,5.599,148.876
C08816=1203.863,9.520,-43.690,-179.637,5.599,148.877
C08817=1203.868,9.270,-43.676,-179.640,5.598,148.878
C08818=1203.873,9.021,-43.662,-179.642,5.598,148.878
C08819=1203.877,8.771,-43.648,-179.645,5.597,148.879
C08820=1203.882,8.521,-43.633,-179.647,5.596,148.879
C08821=1203.888,8.273,-43.618,-179.650,5.596,148.880
C08822=1203.893,8.023,-43.604,-179.653,5.595,148.881
C08823=1203.898,7.773,-43.590,-179.655,5.596,148.881
C08824=1203.903,7.523,-43.575,-179.657,5.595,148.882
C08825=1203.908,7.274,-43.561,-179.660,5.595,148.883
C08826=1203.913,7.024,-43.547,-179.662,5.594,148.883
C08827=1203.919,6.775,-43.533,-179.665,5.593,148.884
C08828=1203.924,6.525,-43.518,-179.667,5.593,148.885
C08829=1203.929,6.276,-43.504,-179.670,5.592,148.885
C08830=1203.934,6.026,-43.490,-179.673,5.592,148.886
C08831=1203.938,5.777,-43.475,-179.675,5.591,148.887
C08832=1203.943,5.527,-43.461,-179.677,5.591,148.887
C08833=1203.949,5.278,-43.447,-179.680,5.591,148.888
C08834=1203.954,5.028,-43.432,-179.682,5.590,148.889
C08835=1203.959,4.779,-43.418,-179.685,5.590,148.889
C08836=1203.964,4.529,-43.404,-179.688,5.589,148.890
C08837=1203.969,4.279,-43.390,-179.690,5.589,148.891
C08838=1203.974,4.030,-43.376,-179.693,5.588,148.891
C08839=1203.979,3.780,-43.361,-179.695,5.587,148.892
C08840=1203.984,3.531,-43.347,-179.697,5.588,148.892
C08841=1203.989,3.261,-43.332,-179.700,5.587,148.893
C08842=1203.995,2.993,-43.316,-179.702,5.587,148.894
C08843=1204.001,2.724,-43.302,-179.705,5.586,148.894
C08844=1204.006,2.454,-43.287,-179.708,5.586,148.895
C08845=1204.011,2.205,-43.273,-179.710,5.585,148.896
C08846=1204.016,1.955,-43.258,-179.713,5.585,148.897
C08847=1204.022,1.706,-43.244,-179.716,5.584,148.897
C08848=1204.026,1.457,-43.231,-179.718,5.584,148.898
C08849=1204.031,1.207,-43.216,-179.721,5.583,148.899
C08850=1204.036,0.957,-43.202,-179.724,5.583,148.899
C08851=1204.041,0.708,-43.188,-179.726,5.582,148.900
C08852=1204.046,0.458,-43.174,-179.728,5.582,148.900
C08853=1204.051,0.208,-43.160,-179.731,5.582,148.901
C08854=1204.056,-0.042,-43.146,-179.733,5.581,148.902
C08855=1204.062,-0.291,-43.132,-179.736,5.581,148.903
C08856=1204.067,-0.540,-43.118,-179.738,5.580,148.903
C08857=1204.071,-0.790,-43.104,-179.741,5.580,148.904
C08858=1204.077,-1.039,-43.090,-179.743,5.579,148.904
C08859=1204.082,-1.288,-43.076,-179.745,5.579,148.905
C08860=1204.087,-1.539,-43.063,-179.748,5.579,148.906
C08861=1204.092,-1.788,-43.048,-179.751,5.578,148.906
C08862=1204.097,-2.037,-43.034,-179.753,5.578,148.907
C08863=1204.102,-2.287,-43.021,-179.756,5.577,148.908
C08864=1204.107,-2.537,-43.006,-179.759,5.577,148.908
C08865=1204.112,-2.786,-42.993,-179.760,5.577,148.909
C08866=1204.117,-3.036,-42.979,-179.763,5.576,148.910
C08867=1204.122,-3.286,-42.965,-179.766,5.576,148.910
C08868=1204.127,-3.534,-42.951,-179.768,5.575,148.911
C08869=1204.132,-3.784,-42.937,-179.771,5.575,148.912
C08870=1204.137,-4.034,-42.923,-179.774,5.574,148.912
C08871=1204.143,-4.283,-42.910,-179.776,5.574,148.913
C08872=1204.148,-4.533,-42.895,-179.778,5.574,148.914
C08873=1204.152,-4.783,-42.882,-179.780,5.573,148.914
C08874=1204.158,-5.032,-42.868,-179.783,5.573,148.915
C08875=1204.163,-5.282,-42.854,-179.786,5.572,148.916
C08876=1204.168,-5.532,-42.840,-179.788,5.572,148.916
C08877=1204.173,-5.781,-42.827,-179.790,5.572,148.917
C08878=1204.178,-6.031,-42.813,-179.793,5.571,148.918
C08879=1204.183,-6.280,-42.799,-179.795,5.571,148.918
C08880=1204.189,-6.530,-42.785,-179.798,5.570,148.919
C08881=1204.193,-6.779,-42.772,-179.801,5.570,148.920
C08882=1204.199,-7.028,-42.758,-179.803,5.569,148.920
C08883=1204.204,-7.279,-42.744,-179.805,5.569,148.921
C08884=1204.208,-7.528,-42.731,-179.808,5.569,148.922
C08885=1204.214,-7.777,-42.717,-179.811,5.568,148.922
C08886=1204.219,-8.027,-42.703,-179.813,5.568,148.923
C08887=1204.224,-8.276,-42.690,-179.815,5.567,148.923
C08888=1204.229,-8.526,-42.676,-179.818,5.567,148.924
C08889=1204.234,-8.776,-42.662,-179.820,5.567,148.925
C08890=1204.239,-9.025,-42.649,-179.823,5.566,148.926
C08891=1204.244,-9.275,-42.635,-179.825,5.566,148.926
C08892=1204.250,-9.524,-42.621,-179.828,5.565,148.927
C08893=1204.254,-9.774,-42.608,-179.830,5.565,148.927
C08894=1204.259,-10.024,-42.594,-179.832,5.565,148.928
C08895=1204.265,-10.274,-42.581,-179.835,5.564,148.929
C08896=1204.269,-10.523,-42.567,-179.838,5.564,148.929
C08897=1204.275,-10.772,-42.553,-179.840,5.563,148.930
C08898=1204.280,-11.022,-42.540,-179.843,5.563,148.931
C08899=1204.285,-11.271,-42.526,-179.845,5.563,148.932
C08900=1204.290,-11.521,-42.513,-179.847,5.562,148.932
C08901=1204.294,-11.771,-42.499,-179.850,5.562,148.933
C08902=1204.300,-12.020,-42.486,-179.853,5.561,148.933
C08903=1204.305,-12.270,-42.472,-179.855,5.561,148.934
C08904=1204.310,-12.519,-42.459,-179.857,5.561,148.935
C08905=1204.315,-12.769,-42.445,-179.860,5.561,148.935
C08906=1204.320,-13.018,-42.432,-179.863,5.560,148.936
C08907=1204.325,-13.269,-42.419,-179.865,5.560,148.937
C08908=1204.331,-13.518,-42.405,-179.867,5.559,148.937
C08909=1204.336,-13.768,-42.392,-179.870,5.559,148.938
C08910=1204.341,-14.017,-42.378,-179.872,5.559,148.939
C08911=1204.346,-14.267,-42.365,-179.875,5.558,148.939
C08912=1204.351,-14.516,-42.351,-179.877,5.558,148.940
C08913=1204.356,-14.766,-42.338,-179.880,5.557,148.941
C08914=1204.362,-15.015,-42.325,-179.882,5.558,148.941
C08915=1204.366,-15.265,-42.311,-179.884,5.557,148.942
C08916=1204.372,-15.514,-42.298,-179.887,5.556,148.943
C08917=1204.376,-15.764,-42.284,-179.890,5.556,148.943
C08918=1204.382,-16.013,-42.271,-179.892,5.555,148.944
C08919=1204.386,-16.264,-42.258,-179.894,5.556,148.945
C08920=1204.392,-16.513,-42.244,-179.897,5.555,148.945
C08921=1204.396,-16.763,-42.231,-179.900,5.555,148.946
C08922=1204.402,-17.012,-42.218,-179.902,5.554,148.947
C08923=1204.406,-17.262,-42.204,-179.905,5.553,148.947
C08924=1204.412,-17.511,-42.191,-179.907,5.554,148.948
C08925=1204.417,-17.761,-42.178,-179.909,5.553,148.949
C08926=1204.422,-18.010,-42.164,-179.912,5.553,148.949
C08927=1204.427,-18.260,-42.151,-179.915,5.552,148.950
C08928=1204.433,-18.510,-42.138,-179.917,5.553,148.951
C08929=1204.437,-18.759,-42.124,-179.919,5.552,148.951
C08930=1204.443,-19.009,-42.111,-179.922,5.551,148.952
C08931=1204.448,-19.258,-42.099,-179.924,5.551,148.953
C08932=1204.453,-19.509,-42.085,-179.927,5.550,148.953
C08933=1204.458,-19.757,-42.072,-179.929,5.551,148.954
C08934=1204.463,-20.007,-42.059,-179.932,5.550,148.955
C08935=1204.468,-20.257,-42.046,-179.934,5.550,148.955
C08936=1204.473,-20.507,-42.033,-179.937,5.549,148.956
C08937=1204.478,-20.756,-42.019,-179.939,5.550,148.957
C08938=1204.484,-21.005,-42.006,-179.941,5.549,148.957
C08939=1204.489,-21.256,-41.992,-179.944,5.548,148.958
C08940=1204.494,-21.505,-41.980,-179.946,5.548,148.959
C08941=1204.499,-21.755,-41.967,-179.949,5.548,148.959
C08942=1204.504,-22.004,-41.953,-179.951,5.548,148.960
C08943=1204.509,-22.253,-41.940,-179.954,5.547,148.961
C08944=1204.514,-22.504,-41.927,-179.957,5.547,148.961
C08945=1204.520,-22.773,-41.914,-179.959,5.546,148.962
C08946=1204.525,-23.042,-41.899,-179.962,5.546,148.963
C08947=1204.530,-23.312,-41.885,-179.964,5.546,148.963
C08948=1204.536,-23.582,-41.871,-179.967,5.545,148.964
C08949=1204.541,-23.831,-41.858,-179.969,5.545,148.965
C08950=1204.546,-24.080,-41.845,-179.972,5.545,148.966
C08951=1204.552,-24.331,-41.832,-179.975,5.544,148.966
C08952=1204.557,-24.579,-41.818,-179.976,5.544,148.967
C08953=1204.562,-24.829,-41.806,-179.979,5.544,148.967
C08954=1204.567,-25.079,-41.792,-179.981,5.543,148.968
C08955=1204.572,-25.328,-41.780,-179.984,5.543,148.969
C08956=1204.577,-25.578,-41.767,-179.986,5.543,148.969
C08957=1204.582,-25.828,-41.754,-179.989,5.542,148.970
C08958=1204.588,-26.077,-41.741,-179.992,5.542,148.971
C08959=1204.592,-26.327,-41.728,-179.994,5.541,148.972
C08960=1204.598,-26.577,-41.715,-179.996,5.541,148.972
C08961=1204.603,-26.826,-41.702,-179.998,5.541,148.973
C08962=1204.608,-27.076,-41.689,179.999,5.541,148.973
C08963=1204.613,-27.326,-41.677,179.996,5.540,148.974
C08964=1204.619,-27.575,-41.663,179.994,5.540,148.975
C08965=1204.623,-27.825,-41.650,179.991,5.540,148.976
C08966=1204.628,-28.075,-41.638,179.989,5.539,148.976
C08967=1204.633,-28.324,-41.625,179.986,5.539,148.977
C08968=1204.639,-28.574,-41.612,179.985,5.539,148.977
C08969=1204.644,-28.824,-41.599,179.982,5.538,148.978
C08970=1204.649,-29.073,-41.586,179.979,5.538,148.979
C08971=1204.654,-29.322,-41.574,179.977,5.538,148.979
C08972=1204.659,-29.572,-41.561,179.975,5.538,148.980
C08973=1204.664,-29.822,-41.548,179.972,5.537,148.981
C08974=1204.669,-30.071,-41.535,179.969,5.537,148.982
C08975=1204.674,-30.321,-41.522,179.968,5.537,148.982
C08976=1204.679,-30.571,-41.510,179.965,5.536,148.983
C08977=1204.684,-30.820,-41.497,179.962,5.536,148.983
C08978=1204.690,-31.069,-41.484,179.960,5.535,148.984
C08979=1204.695,-31.319,-41.471,179.958,5.536,148.985
C08980=1204.700,-31.569,-41.458,179.955,5.535,148.986
C08981=1204.705,-31.819,-41.446,179.952,5.535,148.986
C08982=1204.710,-32.068,-41.434,179.950,5.535,148.987
C08983=1204.716,-32.318,-41.420,179.948,5.534,148.987
C08984=1204.721,-32.568,-41.408,179.945,5.534,148.988
C08985=1204.726,-32.817,-41.395,179.943,5.533,148.989
C08986=1204.731,-33.066,-41.382,179.941,5.534,148.990
C08987=1204.735,-33.316,-41.369,179.938,5.533,148.990
C08988=1204.741,-33.566,-41.357,179.935,5.533,148.991
C08989=1204.746,-33.816,-41.345,179.933,5.532,148.992
C08990=1204.752,-34.065,-41.332,179.931,5.533,148.992
C08991=1204.756,-34.315,-41.319,179.928,5.532,148.993
C08992=1204.762,-34.565,-41.306,179.926,5.531,148.993
C08993=1204.767,-34.815,-41.294,179.924,5.532,148.994
C08994=1204.772,-35.064,-41.282,179.921,5.531,148.995
C08995=1204.777,-35.313,-41.269,179.918,5.531,148.996
C08996=1204.782,-35.563,-41.256,179.916,5.530,148.996
C08997=1204.787,-35.812,-41.243,179.914,5.531,148.997
C08998=1204.792,-36.062,-41.232,179.911,5.530,148.998
C08999=1204.797,-36.312,-41.219,179.909,5.529,148.998
C09000=1204.803,-36.561,-41.206,179.907,5.530,148.999
C09001=1204.808,-36.811,-41.193,179.904,5.529,149.000
C09002=1204.813,-37.061,-41.181,179.901,5.529,149.000
C09003=1204.818,-37.311,-41.168,179.899,5.529,149.001
C09004=1204.823,-37.560,-41.156,179.897,5.529,149.002
C09005=1204.829,-37.810,-41.144,179.894,5.528,149.002
C09006=1204.834,-38.059,-41.131,179.892,5.527,149.003
C09007=1204.839,-38.309,-41.118,179.890,5.528,149.004
C09008=1204.844,-38.559,-41.106,179.887,5.527,149.004
C09009=1204.849,-38.808,-41.094,179.884,5.527,149.005
C09010=1204.854,-39.058,-41.081,179.882,5.527,149.006
C09011=1204.859,-39.307,-41.069,179.880,5.527,149.006
C09012=1204.865,-39.557,-41.057,179.877,5.526,149.007
C09013=1204.869,-39.807,-41.044,179.875,5.526,149.008
C09014=1204.875,-40.057,-41.032,179.873,5.526,149.008
C09015=1204.880,-40.306,-41.019,179.870,5.525,149.009
C09016=1204.885,-40.556,-41.007,179.867,5.525,149.010
C09017=1204.890,-40.806,-40.995,179.865,5.525,149.010
C09018=1204.896,-41.055,-40.982,179.863,5.525,149.011
C09019=1204.901,-41.304,-40.970,179.860,5.524,149.012
C09020=1204.906,-41.554,-40.958,179.858,5.524,149.012
C09021=1204.911,-41.804,-40.945,179.856,5.524,149.013
C09022=1204.916,-42.054,-40.933,179.853,5.523,149.014
C09023=1204.921,-42.303,-40.920,179.851,5.523,149.014
C09024=1204.927,-42.553,-40.908,179.848,5.523,149.015
C09025=1204.932,-42.803,-40.896,179.846,5.523,149.016
C09026=1204.936,-43.052,-40.884,179.843,5.523,149.016
C09027=1204.942,-43.302,-40.872,179.841,5.522,149.017
C09028=1204.947,-43.551,-40.859,179.838,5.522,149.018
C09029=1204.952,-43.801,-40.847,179.837,5.522,149.018
C09030=1204.957,-44.051,-40.834,179.834,5.521,149.019
C09031=1204.962,-44.301,-40.823,179.831,5.521,149.020
C09032=1204.967,-44.550,-40.810,179.829,5.521,149.020
C09033=1204.973,-44.800,-40.798,179.826,5.521,149.021
C09034=1204.978,-45.049,-40.785,179.824,5.520,149.022
C09035=1204.983,-45.299,-40.774,179.821,5.520,149.022
C09036=1204.988,-45.549,-40.761,179.820,5.520,149.023
C09037=1204.993,-45.798,-40.750,179.817,5.519,149.024
C09038=1204.998,-46.048,-40.737,179.814,5.519,149.024
C09039=1205.004,-46.298,-40.725,179.812,5.519,149.025
C09040=1205.009,-46.547,-40.713,179.809,5.519,149.026
C09041=1205.014,-46.797,-40.701,179.807,5.518,149.026
C09042=1205.019,-47.047,-40.689,179.805,5.519,149.027
C09043=1205.025,-47.296,-40.676,179.802,5.518,149.028
C09044=1205.029,-47.546,-40.665,179.800,5.517,149.028
C09045=1205.034,-47.795,-40.652,179.798,5.518,149.029
C09046=1205.040,-48.045,-40.640,179.795,5.517,149.030
C09047=1205.045,-48.295,-40.629,179.792,5.517,149.030
C09048=1205.050,-48.544,-40.616,179.790,5.517,149.031
C09049=1205.056,-48.815,-40.603,179.788,5.517,149.032
C09050=1205.061,-49.085,-40.590,179.785,5.516,149.033
C09051=1205.067,-49.355,-40.577,179.782,5.516,149.033
C09052=1205.072,-49.625,-40.564,179.780,5.516,149.034
C09053=1205.077,-49.874,-40.552,179.778,5.516,149.035
C09054=1205.083,-50.124,-40.540,179.775,5.515,149.035
C09055=1205.088,-50.374,-40.528,179.773,5.516,149.036
C09056=1205.093,-50.623,-40.516,179.770,5.515,149.037
C09057=1205.098,-50.873,-40.504,179.768,5.515,149.037
C09058=1205.103,-51.123,-40.492,179.766,5.515,149.038
C09059=1205.109,-51.372,-40.480,179.763,5.514,149.039
C09060=1205.113,-51.622,-40.468,179.761,5.514,149.039
C09061=1205.119,-51.872,-40.457,179.759,5.514,149.040
C09062=1205.124,-52.121,-40.444,179.756,5.514,149.041
C09063=1205.129,-52.371,-40.432,179.753,5.513,149.041
C09064=1205.134,-52.621,-40.421,179.751,5.514,149.042
C09065=1205.139,-52.871,-40.409,179.749,5.513,149.043
C09066=1205.145,-53.120,-40.396,179.746,5.512,149.043
C09067=1205.149,-53.370,-40.385,179.744,5.513,149.044
C09068=1205.155,-53.620,-40.373,179.742,5.512,149.045
C09069=1205.160,-53.869,-40.361,179.739,5.512,149.045
C09070=1205.165,-54.119,-40.349,179.737,5.512,149.046
C09071=1205.170,-54.368,-40.337,179.734,5.512,149.047
C09072=1205.175,-54.618,-40.325,179.733,5.512,149.047
C09073=1205.181,-54.868,-40.314,179.730,5.511,149.048
C09074=1205.186,-55.117,-40.302,179.727,5.511,149.049
C09075=1205.191,-55.367,-40.290,179.725,5.511,149.049
C09076=1205.197,-55.616,-40.278,179.722,5.511,149.050
C09077=1205.201,-55.866,-40.267,179.720,5.510,149.051
C09078=1205.207,-56.116,-40.255,179.718,5.511,149.052
C09079=1205.212,-56.366,-40.243,179.716,5.510,149.052
C09080=1205.217,-56.615,-40.231,179.713,5.509,149.053
C09081=1205.222,-56.865,-40.219,179.711,5.510,149.053
C09082=1205.227,-57.115,-40.208,179.708,5.509,149.054
C09083=1205.232,-57.364,-40.196,179.705,5.509,149.055
C09084=1205.238,-57.614,-40.184,179.703,5.509,149.056
C09085=1205.242,-57.864,-40.173,179.701,5.508,149.056
C09086=1205.248,-58.113,-40.161,179.699,5.509,149.057
C09087=1205.254,-58.363,-40.149,179.696,5.508,149.057
C09088=1205.258,-58.612,-40.137,179.694,5.508,149.058
C09089=1205.263,-58.862,-40.126,179.692,5.508,149.059
C09090=1205.268,-59.112,-40.114,179.689,5.508,149.060
C09091=1205.274,-59.362,-40.102,179.686,5.507,149.060
C09092=1205.278,-59.611,-40.091,179.685,5.507,149.061
C09093=1205.284,-59.861,-40.079,179.682,5.507,149.061
C09094=1205.290,-60.110,-40.068,179.680,5.507,149.062
C09095=1205.294,-60.360,-40.056,179.677,5.507,149.063
C09096=1205.300,-60.610,-40.044,179.675,5.506,149.064
C09097=1205.305,-60.860,-40.033,179.673,5.507,149.064
C09098=1205.310,-61.110,-40.021,179.670,5.506,149.065
C09099=1205.315,-61.359,-40.010,179.668,5.505,149.065
C09100=1205.320,-61.609,-39.998,179.666,5.506,149.066
C09101=1205.325,-61.858,-39.987,179.663,5.505,149.067
C09102=1205.331,-62.108,-39.975,179.661,5.506,149.068
C09103=1205.336,-62.358,-39.963,179.658,5.505,149.068
C09104=1205.341,-62.608,-39.952,179.656,5.505,149.069
C09105=1205.346,-62.858,-39.940,179.654,5.505,149.069
C09106=1205.351,-63.107,-39.929,179.651,5.504,149.070
C09107=1205.357,-63.356,-39.917,179.649,5.504,149.071
C09108=1205.362,-63.606,-39.906,179.647,5.504,149.072
C09109=1205.367,-63.856,-39.894,179.644,5.504,149.072
C09110=1205.372,-64.106,-39.883,179.642,5.504,149.073
C09111=1205.377,-64.356,-39.871,179.639,5.504,149.074
C09112=1205.383,-64.604,-39.860,179.637,5.503,149.074
C09113=1205.387,-64.854,-39.849,179.635,5.503,149.075
C09114=1205.393,-65.104,-39.837,179.632,5.503,149.076
C09115=1205.398,-65.354,-39.826,179.630,5.503,149.076
C09116=1205.403,-65.604,-39.815,179.627,5.503,149.077
C09117=1205.408,-65.853,-39.804,179.625,5.502,149.078
C09118=1205.414,-66.103,-39.792,179.623,5.502,149.078
C09119=1205.419,-66.353,-39.780,179.621,5.502,149.079
C09120=1205.424,-66.603,-39.769,179.618,5.502,149.080
C09121=1205.429,-66.852,-39.757,179.616,5.502,149.080
C09122=1205.435,-67.101,-39.746,179.613,5.501,149.081
C09123=1205.440,-67.352,-39.735,179.611,5.501,149.082
C09124=1205.444,-67.601,-39.724,179.609,5.501,149.082
C09125=1205.450,-67.851,-39.712,179.607,5.501,149.083
C09126=1205.455,-68.100,-39.701,179.604,5.501,149.084
C09127=1205.461,-68.350,-39.689,179.601,5.500,149.084
C09128=1205.465,-68.600,-39.678,179.599,5.500,149.085
C09129=1205.470,-68.850,-39.667,179.597,5.500,149.086
C09130=1205.476,-69.099,-39.656,179.595,5.500,149.086
C09131=1205.481,-69.349,-39.645,179.592,5.500,149.087
C09132=1205.486,-69.599,-39.633,179.590,5.499,149.088
C09133=1205.492,-69.848,-39.622,179.588,5.500,149.088
C09134=1205.497,-70.098,-39.611,179.585,5.499,149.089
C09135=1205.502,-70.348,-39.599,179.583,5.499,149.090
C09136=1205.507,-70.598,-39.588,179.581,5.499,149.090
C09137=1205.512,-70.846,-39.577,179.578,5.498,149.091
C09138=1205.518,-71.097,-39.566,179.576,5.499,149.092
C09139=1205.523,-71.347,-39.555,179.573,5.498,149.092
C09140=1205.529,-71.596,-39.543,179.571,5.498,149.093
C09141=1205.534,-71.846,-39.532,179.569,5.498,149.094
C09142=1205.538,-72.096,-39.521,179.566,5.497,149.094
C09143=1205.544,-72.346,-39.509,179.564,5.498,149.095
